# B&R Automation Studio project KeePak_BlissNewScreen (part 2)

#### Cyclic1.st
```iecst
PROGRAM _CYCLIC
	(* Insert code here *)

    // HMI Glue pattern inputs are in inches, but the code needs mm
    gAdhesiveCtrlInterface.Parameters.AdhesivePatterns[0].DelayDistance[0] := gAdhesiveCtrlInterface.Parameters.AdhesiveHMIPatterns[0].DelayDistance[0] * 25.4;
    gAdhesiveCtrlInterface.Parameters.AdhesivePatterns[0].DelayDistance[1] := gAdhesiveCtrlInterface.Parameters.AdhesiveHMIPatterns[0].DelayDistance[1] * 25.4;
    gAdhesiveCtrlInterface.Parameters.AdhesivePatterns[0].DelayDistance[2] := gAdhesiveCtrlInterface.Parameters.AdhesiveHMIPatterns[0].DelayDistance[2] * 25.4;
    gAdhesiveCtrlInterface.Parameters.AdhesivePatterns[0].DelayDistance[3] := gAdhesiveCtrlInterface.Parameters.AdhesiveHMIPatterns[0].DelayDistance[3] * 25.4;
    gAdhesiveCtrlInterface.Parameters.AdhesivePatterns[1].DelayDistance[0] := gAdhesiveCtrlInterface.Parameters.AdhesiveHMIPatterns[1].DelayDistance[0] * 25.4;
    gAdhesiveCtrlInterface.Parameters.AdhesivePatterns[1].DelayDistance[1] := gAdhesiveCtrlInterface.Parameters.AdhesiveHMIPatterns[1].DelayDistance[1] * 25.4;
    gAdhesiveCtrlInterface.Parameters.AdhesivePatterns[1].DelayDistance[2] := gAdhesiveCtrlInterface.Parameters.AdhesiveHMIPatterns[1].DelayDistance[2] * 25.4;
    gAdhesiveCtrlInterface.Parameters.AdhesivePatterns[1].DelayDistance[3] := gAdhesiveCtrlInterface.Parameters.AdhesiveHMIPatterns[1].DelayDistance[3] * 25.4;
    gAdhesiveCtrlInterface.Parameters.AdhesivePatterns[2].DelayDistance[0] := gAdhesiveCtrlInterface.Parameters.AdhesiveHMIPatterns[2].DelayDistance[0] * 25.4;
    gAdhesiveCtrlInterface.Parameters.AdhesivePatterns[2].DelayDistance[1] := gAdhesiveCtrlInterface.Parameters.AdhesiveHMIPatterns[2].DelayDistance[1] * 25.4;
    gAdhesiveCtrlInterface.Parameters.AdhesivePatterns[2].DelayDistance[2] := gAdhesiveCtrlInterface.Parameters.AdhesiveHMIPatterns[2].DelayDistance[2] * 25.4;
    gAdhesiveCtrlInterface.Parameters.AdhesivePatterns[2].DelayDistance[3] := gAdhesiveCtrlInterface.Parameters.AdhesiveHMIPatterns[2].DelayDistance[3] * 25.4;
    gAdhesiveCtrlInterface.Parameters.AdhesivePatterns[3].DelayDistance[0] := gAdhesiveCtrlInterface.Parameters.AdhesiveHMIPatterns[3].DelayDistance[0] * 25.4;
    gAdhesiveCtrlInterface.Parameters.AdhesivePatterns[3].DelayDistance[1] := gAdhesiveCtrlInterface.Parameters.AdhesiveHMIPatterns[3].DelayDistance[1] * 25.4;
    gAdhesiveCtrlInterface.Parameters.AdhesivePatterns[3].DelayDistance[2] := gAdhesiveCtrlInterface.Parameters.AdhesiveHMIPatterns[3].DelayDistance[2] * 25.4;
    gAdhesiveCtrlInterface.Parameters.AdhesivePatterns[3].DelayDistance[3] := gAdhesiveCtrlInterface.Parameters.AdhesiveHMIPatterns[3].DelayDistance[3] * 25.4;

    gAdhesiveCtrlInterface.Parameters.AdhesivePatterns[0].GlueOnDistance[0] := gAdhesiveCtrlInterface.Parameters.AdhesiveHMIPatterns[0].GlueOnDistance[0] * 25.4;
    gAdhesiveCtrlInterface.Parameters.AdhesivePatterns[0].GlueOnDistance[1] := gAdhesiveCtrlInterface.Parameters.AdhesiveHMIPatterns[0].GlueOnDistance[1] * 25.4;
    gAdhesiveCtrlInterface.Parameters.AdhesivePatterns[0].GlueOnDistance[2] := gAdhesiveCtrlInterface.Parameters.AdhesiveHMIPatterns[0].GlueOnDistance[2] * 25.4;
    gAdhesiveCtrlInterface.Parameters.AdhesivePatterns[0].GlueOnDistance[3] := gAdhesiveCtrlInterface.Parameters.AdhesiveHMIPatterns[0].GlueOnDistance[3] * 25.4;
    gAdhesiveCtrlInterface.Parameters.AdhesivePatterns[1].GlueOnDistance[0] := gAdhesiveCtrlInterface.Parameters.AdhesiveHMIPatterns[1].GlueOnDistance[0] * 25.4;
    gAdhesiveCtrlInterface.Parameters.AdhesivePatterns[1].GlueOnDistance[1] := gAdhesiveCtrlInterface.Parameters.AdhesiveHMIPatterns[1].GlueOnDistance[1] * 25.4;
    gAdhesiveCtrlInterface.Parameters.AdhesivePatterns[1].GlueOnDistance[2] := gAdhesiveCtrlInterface.Parameters.AdhesiveHMIPatterns[1].GlueOnDistance[2] * 25.4;
    gAdhesiveCtrlInterface.Parameters.AdhesivePatterns[1].GlueOnDistance[3] := gAdhesiveCtrlInterface.Parameters.AdhesiveHMIPatterns[1].GlueOnDistance[3] * 25.4;
    gAdhesiveCtrlInterface.Parameters.AdhesivePatterns[2].GlueOnDistance[0] := gAdhesiveCtrlInterface.Parameters.AdhesiveHMIPatterns[2].GlueOnDistance[0] * 25.4;
    gAdhesiveCtrlInterface.Parameters.AdhesivePatterns[2].GlueOnDistance[1] := gAdhesiveCtrlInterface.Parameters.AdhesiveHMIPatterns[2].GlueOnDistance[1] * 25.4;
    gAdhesiveCtrlInterface.Parameters.AdhesivePatterns[2].GlueOnDistance[2] := gAdhesiveCtrlInterface.Parameters.AdhesiveHMIPatterns[2].GlueOnDistance[2] * 25.4;
    gAdhesiveCtrlInterface.Parameters.AdhesivePatterns[2].GlueOnDistance[3] := gAdhesiveCtrlInterface.Parameters.AdhesiveHMIPatterns[2].GlueOnDistance[3] * 25.4;
    gAdhesiveCtrlInterface.Parameters.AdhesivePatterns[3].GlueOnDistance[0] := gAdhesiveCtrlInterface.Parameters.AdhesiveHMIPatterns[3].GlueOnDistance[0] * 25.4;
    gAdhesiveCtrlInterface.Parameters.AdhesivePatterns[3].GlueOnDistance[1] := gAdhesiveCtrlInterface.Parameters.AdhesiveHMIPatterns[3].GlueOnDistance[1] * 25.4;
    gAdhesiveCtrlInterface.Parameters.AdhesivePatterns[3].GlueOnDistance[2] := gAdhesiveCtrlInterface.Parameters.AdhesiveHMIPatterns[3].GlueOnDistance[2] * 25.4;
    gAdhesiveCtrlInterface.Parameters.AdhesivePatterns[3].GlueOnDistance[3] := gAdhesiveCtrlInterface.Parameters.AdhesiveHMIPatterns[3].GlueOnDistance[3] * 25.4;

    //SAFETY CHECKS 0001
    IF NOT gAlarmSystemActive THEN
        RETURN;
    END_IF

    //AIR PRESSURE ON/NOK 0002
    //Do not set air pressure alarm unless air pressure has been low for 20 seconds
    AirPressureNotOKTimer.PT := T#20s;
    AirPressureNotOKTimer.IN := (NOT gIO.DIs.AirPressureOK AND NOT gIsSimulated);
    AirPressureNotOKTimer();
    AirPressureNotOK         := AirPressureNotOKTimer.Q;

    //MP ALARMX CHECK STATE AIR PRESSURE LOW 0003
    AirPressureAlarmActive := MpAlarmXCheckState(gAlarmXCore, ALARM_AIR_PRESSURE_LOW, mpALARMX_STATE_ACTIVE);

    //MP ALARMX SET/RESET AIR PRESSURE LOW 0004 AND 0005
    //Set/clear air pressure alarm
    IF (AirPressureNotOK AND NOT AirPressureAlarmActive) THEN
        status := MpAlarmXSet(gAlarmXCore,ALARM_AIR_PRESSURE_LOW);
    ELSIF (NOT AirPressureNotOK AND AirPressureAlarmActive) THEN
        status := MpAlarmXReset(gAlarmXCore,ALARM_AIR_PRESSURE_LOW);
    END_IF

    //MP ALARMX CHECK STATE SAFETY OK/NOK 0006
    SafetyNotOKActive := MpAlarmXCheckState(gAlarmXCore, ALARM_SAFETY_NOTOK, mpALARMX_STATE_ACTIVE);

    //MP ALARMX SET/RESET SAFETY OK/NOK 0007 AND 0008
    //Set/Clear Safety Alarm
    IF (NOT gIO.DIs.SafetyOK AND NOT SafetyNotOKActive AND gIO.SafetyStatus.SafetyProgramRunning) THEN
        status := MpAlarmXSet(gAlarmXCore,ALARM_SAFETY_NOTOK);
    ELSIF (gIO.DIs.SafetyOK AND SafetyNotOKActive AND gIO.SafetyStatus.SafetyProgramRunning) THEN
        status := MpAlarmXReset(gAlarmXCore,ALARM_SAFETY_NOTOK);
    END_IF

    //MP ALARMX CHECK STATE GUARD DOOR 0009
    GuardDoorNotOKActive := MpAlarmXCheckState(gAlarmXCore, ALARM_SAFETY_GUARD_DOOR, mpALARMX_STATE_ACTIVE);

    //MP ALARMX SET/RESET GUARD DOORS 0010 AND 0011
    //Set/Clear Safety Alarm
    IF (NOT gIO.SafetyStatus.GuardDoorsOK AND NOT GuardDoorNotOKActive AND gIO.SafetyStatus.SafetyProgramRunning) THEN
        status := MpAlarmXSet(gAlarmXCore,ALARM_SAFETY_GUARD_DOOR);
    ELSIF (gIO.SafetyStatus.GuardDoorsOK AND GuardDoorNotOKActive AND gIO.SafetyStatus.SafetyProgramRunning) THEN
        status := MpAlarmXReset(gAlarmXCore,ALARM_SAFETY_GUARD_DOOR);
    END_IF

    //MP ALARMX CHECK STATE FRONT ESTOP 0012
    FrontEStopNotOKActive := MpAlarmXCheckState(gAlarmXCore, ALARM_SAFETY_FRONT_ESTOP, mpALARMX_STATE_ACTIVE);

    //MP ALARMX SET/RESET FRONT ESTOP 0013 AND 0014
    //Set/Clear Safety Alarm
    IF (NOT gIO.SafetyStatus.FrontEStopOK AND NOT FrontEStopNotOKActive AND gIO.SafetyStatus.SafetyProgramRunning) THEN
        status := MpAlarmXSet(gAlarmXCore,ALARM_SAFETY_FRONT_ESTOP);
    ELSIF (gIO.SafetyStatus.FrontEStopOK AND FrontEStopNotOKActive AND gIO.SafetyStatus.SafetyProgramRunning) THEN
        status := MpAlarmXReset(gAlarmXCore,ALARM_SAFETY_FRONT_ESTOP);
    END_IF

    //MP ALARMX CHECK STATE REAR ESTOP 0015
    RearEStopNotOKActive := MpAlarmXCheckState(gAlarmXCore, ALARM_SAFETY_REAR_ESTOP, mpALARMX_STATE_ACTIVE);

    //MP ALARMX SET/RESET REAR ESTOP 0016 AND 0017
    //Set/Clear Safety Alarm
    IF (NOT gIO.SafetyStatus.BackEstopOK AND NOT RearEStopNotOKActive AND gIO.SafetyStatus.SafetyProgramRunning) THEN
        status := MpAlarmXSet(gAlarmXCore,ALARM_SAFETY_REAR_ESTOP);
    ELSIF (gIO.SafetyStatus.BackEstopOK AND RearEStopNotOKActive AND gIO.SafetyStatus.SafetyProgramRunning) THEN
        status := MpAlarmXReset(gAlarmXCore,ALARM_SAFETY_REAR_ESTOP);
    END_IF

    //TURN AIR ON 0018
    //If safety is OK, Turn air On and turn off the red light
    gIO.DOs.AirOn         := gIO.DIs.SafetyOK;
    gIO.DOs.RedLightStack := NOT (gIO.DIs.SafetyOK AND NOT gModeControlInterface.Status.BlissPanelAlarmActive);

    //NO ALARMS GREEN LIGHT 0019
    //If there are no alarms active, turn on the green light
    gIO.DOs.GreenLightStack := NOT gAlarmActive;

    //ALARM YELLOW LIGHT 0020
    //If there is an active alarm, or the hopper is low, turn on yellow stack light
    gIO.DOs.AmberLightStack := (gAlarmActive OR gIO.DIs.BodyHopperLow);

	//DO NOT FINISH CYCLE OF ANYTHING OTHER THAN STOP BUTTON IS PRESSED 0024
	//If an alarm is active or safety is not ok or jog mode is selected, do not finish the selected cycle
	IF (gServoFeedInterface.Status.Error OR gBodyHopperInterface.Status.Error OR gLeftHopperInterface.Status.Error OR gRightHopperInterface.Status.Error OR gServoRamInterface.Status.Error OR
		NOT gIO.DIs.SafetyOK OR gHMI.Commands.SelectJogMode OR gHighSeverityAlarmActive OR BodyCheckError) THEN
		PickAndPlaceHasBox                         := FALSE;
		PickAndPlaceDwelling                       := FALSE;
		PhotoEyeSeen                               := FALSE;
		Vacuum_ON                                  := FALSE;
		gIO.DOs.X_PickSolenoid                     := FALSE;
		gIO.DOs.BlowOffOn                          := FALSE;
	END_IF

	//DOES NOT LET MACHINE RUN IF GLUE SYSTEM HAS AN ERROR 0025
	//Do not allow machine to run if glue system has an alarm (Removed gLowSeverityAlarmActive)
	IF (gAdhesiveCtrlInterface.Status.AlarmActive OR
		gServoFeedInterface.Status.Error OR gBodyHopperInterface.Status.Error OR gLeftHopperInterface.Status.Error OR gRightHopperInterface.Status.Error OR gServoRamInterface.Status.Error OR
		gLowSeverityAlarmActive OR gHighSeverityAlarmActive OR gServoPnPInterface.Status.Error) THEN
		gHMI.Commands.RequestVFDRun := FALSE;
	END_IF

	//AUTO MODE RUN REQUEST FINISH CYCLE 0026
	//If we're in auto mode, and run request has been made or we should finish the running, set move request
	MoveVelocityRequest := (gHMI.Commands.SelectAutoMode AND gHMI.Commands.RequestVFDRun);

	//RAM POSITION AND STOP POSITION (360-0 ROLLOVER)DetermineDistanceToStopPos 0027
	DistanceFromStopPosition := DetermineDistanceToStopPos(gIO.Encoders.FeedEncoderPos, gModeControlInterface.Parameters.StopPosition);

	//KEEPS SERVOS RUNNING TO FINISH CYCLE 0030
	//VFD run command was the run command for the old machine. Keep servos cycling while it is true
	gHMI.Commands.StartBodyHopper := gHMI.Commands.RequestVFDRun;
	gHMI.Commands.StartLeftHopper := gHMI.Commands.RequestVFDRun;
	gHMI.Commands.StartRightHopper := gHMI.Commands.RequestVFDRun;
	gHMI.Commands.StartServoFeed   := (gHMI.Commands.RequestVFDRun (*AND NOT DownstreamBlocked*) AND NOT StopFeedServo);
	gHMI.Commands.CycleServoRam    := gHMI.Commands.RequestVFDRun;
	gHMI.Commands.CycleServoPnP    := gHMI.Commands.RequestVFDRun;
	// The discharge conveyor is controlled by three bits.
	// If #1 is on, then it is running slow. If #1 and #3 are on, then it is running medium speed. #2 Can be used if we need a faster speed.
	gIO.DOs.OutConveyorOn_1 := gHMI.Commands.RequestVFDRun OR (gCyclesToFinish > 0);
	gIO.DOs.OutConveyorOn_2 := gHMI.Commands.RequestVFDRun OR (gCyclesToFinish > 0);
	gIO.DOs.OutConveyorOn_3 := gHMI.Commands.RequestVFDRun OR (gCyclesToFinish > 0);

	//RISING EDGE FOR SERVOINPUT SIGNAL 0031
	Rtrig_FeedServoTMR(CLK := FeedServoTMR.Q);
	StopFeed := Rtrig_FeedServoTMR.Q;

	//0032 SERVO RAM TRIGGER SET IN FEED HANDLER. COMMENTED OUT

	//HOPPER LOW ALARMS 0033
	BodyHopperLowTMR.IN := gIO.DIs.BodyHopperLow;
    BodyHopperLowTMR.PT := gHMI.Parameters.LowBodyHopperTime;
    BodyHopperLowTMR();
    IF BodyHopperLowTMR.Q THEN
        BodyHopperLowAlarm := TRUE;
	END_IF
	LeftHopperLowTMR.IN := gIO.DIs.LeftHopperLow;
	LeftHopperLowTMR.PT := gHMI.Parameters.LowLeftHopperTime;
	LeftHopperLowTMR();
	IF LeftHopperLowTMR.Q THEN
		LeftHopperLowAlarm := TRUE;
	END_IF
	RightHopperLowTMR.IN := gIO.DIs.RightHopperLow;
	RightHopperLowTMR.PT := gHMI.Parameters.LowRightHopperTime;
	RightHopperLowTMR();
	IF RightHopperLowTMR.Q THEN
		RightHopperLowAlarm := TRUE;
	END_IF

    //FEED STOP TIMER 0034
    //Timer for the HopperLows to trigger StopFeed
    FeedStopTimer.IN := gIO.DIs.BodyHopperLow OR gIO.DIs.RightHopperLow OR gIO.DIs.LeftHopperLow;
    FeedStopTimer.PT := gHMI.Parameters.LowHopperTime;
    FeedStopTimer();
    HoperLowStop     := FeedStopTimer.Q;

    //HOPPER LOW ALARM RESET 0035
    IF NOT gIO.DIs.BodyHopperLow THEN
        BodyHopperLowAlarm := FALSE;
	END_IF
	IF NOT gIO.DIs.LeftHopperLow THEN
		LeftHopperLowAlarm := FALSE;
	END_IF
	IF NOT gIO.DIs.RightHopperLow THEN
		RightHopperLowAlarm := FALSE;
	END_IF

	//==========================================================================================================================================================
	//==========================================================================================================================================================

	//PHOTO EYES SETTING AND RESETTING
	IF (gIO.DIs.AdhesivePhotoEye) THEN
		PhotoEyeSeen := TRUE;
	END_IF
    IF gIO.DIs.BodyDetect THEN
        PhotoEyeSeen := FALSE;
    END_IF

    //0047
    //Latch the encoder position. this marks the start of the glue cycle
    Rtrig_PhotoEyeSeen(CLK := PhotoEyeSeen);
    IF (Rtrig_PhotoEyeSeen.Q AND ((gHMI.Commands.SelectAutoMode AND gHMI.Commands.RequestVFDRun) OR (gCyclesToFinish > 0))) THEN
        gAdhesiveCtrlInterface.Status.LatchedEncoderPos := LREAL_TO_REAL(gServoFeedInterface.Status.ActualPosition);
        DistanceAfterLatch                              := 0;
        OldEncoderPos                                   := LREAL_TO_REAL(gServoFeedInterface.Status.ActualPosition);
    END_IF

    //0048
    //Determine how far the ram has moved since the photo eye was last seen
    DistanceAfterLatch := (ComputeDistanceMoved(LREAL_TO_REAL(gServoFeedInterface.Status.ActualPosition),OldEncoderPos) + DistanceAfterLatch);

    //0049
    OldEncoderPos := LREAL_TO_REAL(gServoFeedInterface.Status.ActualPosition);

	//BODY PANEL TIMEOUT 0052
	//If the machine is running and a box has passed the photoeyes, but hasn't cleared the photo eye for LowFeedJamTime amount of time, then raise an alarm
    BodyPanelTimeout.PT := gHMI.Parameters.LowFeedJamTime;
    BodyPanelTimeout.IN := (gHMI.Commands.RequestVFDRun AND gIO.DIs.BodyDetect);
    BodyPanelTimeout();
    IF BodyPanelTimeout.Q THEN
        BodyCheckError := TRUE;
    ELSIF gHMI.Commands.RequestReset THEN
        BodyCheckError := FALSE;
	END_IF

	//INFEED TIMEOUT
	//If the machine is running and a box hasnt passed the photoeyes for LowFeedJamTime amount of time, then raise an alarm
	InfeedTimeout.PT := gHMI.Parameters.TopFeedJamTime;
	InfeedTimeout.IN := (gHMI.Commands.RequestVFDRun AND NOT gIO.DIs.BodyDetect);
	InfeedTimeout();
	IF InfeedTimeout.Q THEN
		InfeedCheckError := TRUE;
	ELSIF gHMI.Commands.RequestReset THEN
		InfeedCheckError := FALSE;
	END_IF

    //0053 AND 0054 LUBE COUNTER
    LubricationOK := (LubeCount < gHMI.Parameters.SetCycleCount);

    Rtrig_LubricationCounter(CLK := gIO.DIs.LubricationCounter);
    LubricationCounter.CU    := Rtrig_LubricationCounter.Q;
    LubricationCounter.RESET := LubeReset;
    LubricationCounter.PV    := UDINT_TO_UINT(gHMI.Parameters.LubeCycleCount);
    LubricationCounter();
    CountReset               := LubricationCounter.Q;

    //0055 COUNT AND LUBE COUNT RESET
    LubeReset := CountReset;
    IF CountReset THEN
        LubeCount := 0;
	END_IF

	//make it a fault if the system is reuqested to run while any hopper is off
	IF gHMI.Commands.RequestVFDRun AND (gIO.DIs.LeftHopperMotor_OFF OR gIO.DIs.RightHopperMotor_OFF OR gIO.DIs.BodyHopperMotor_OFF) THEN
		HopperRunningError := TRUE;
	ELSIF gHMI.Commands.RequestReset THEN
		HopperRunningError := FALSE;
	END_IF

    //Disabled this due to the error triggering and not clearing after a few hours
//    PnPTimeout.PT := T#3600s;
//    PnPTimeout.IN := NOT gHMI.Commands.RequestVFDRun AND (gHMI.Commands.RequestStop OR gServoPnPInterface.Status.PoweredOn);
//    PnPTimeout();
 //   IF PnPTimeout.Q THEN
//        PnPTimeoutError := TRUE;
//    ELSIF gHMI.Commands.RequestReset THEN
//        PnPTimeoutError := FALSE;
//    END_IF

	END_PROGRAM
```

### Variables.var
```iecst
VAR
	StartDwellTimer : TON;
	AtTorqueTimer : TON;
	state : ServoHopperState_enum;
END_VAR
VAR RETAIN
	CycleCount : UDINT;
END_VAR
VAR
	ResetTimeoutAlarm : BOOL;
	ResetTimeoutTimer : TON;
END_VAR
```

### Program Logical/ServoMotion/LeftHopperHandler

#### Main.st
```iecst
PROGRAM _INIT
	(* Insert code here *)

	gHMI.Parameters.LeftHopperJogVelocity := 3.35;
	gHMI.Parameters.LeftHopperVelocity := 3.35;
	gHMI.Parameters.LeftHopperAccel := 180.0;

	gHMI.Parameters.LeftHopperTorqueLimit := 1.0;

	gHMI.Parameters.LeftHopperDwellTime := 1500; //1 s
	gHMI.Parameters.AtTorqueTime := 500; //1 s

	gHMI.Parameters.LeftHopperTimeoutTime := 600000; //10 minutes

END_PROGRAM

PROGRAM _CYCLIC

	IF gNumActiveAlarms  > 0 THEN
		state := SERVOHOPPER_ERROR;
	END_IF

	IF gHighSeverityAlarmActive THEN
		state := SERVOHOPPER_ERROR;
	END_IF

	//make sure that torque limiting is turned on while jogging
	//	IF EDGEPOS(gHMI.Commands.JogLeftHopperPos) THEN
	//		gLeftHopperInterface.Commands.ToMapp.TorqueLimitingOn := TRUE;
	//	END_IF
	//	IF EDGEPOS(gHMI.Commands.JogLeftHopperNeg) THEN
	//		gLeftHopperInterface.Commands.ToMapp.TorqueLimitingOn := TRUE;
	//	END_IF

	StartDwellTimer.IN := FALSE; //clear otuside state machine. will be set true in appropriate state
	AtTorqueTimer.IN := FALSE;
	ResetTimeoutTimer.IN := FALSE;

	// If the hopper has been reset but the machine isn't running, only let the hopper run for an alotted time to protect the motor
	IF gIO.DIs.LeftHopperMotor_RUN AND NOT gLeftHopperInterface.Status.Error AND (NOT gHMI.Commands.RequestVFDRun) THEN
		ResetTimeoutTimer.IN := TRUE;
	END_IF
	IF ResetTimeoutTimer.Q THEN
		ResetTimeoutAlarm := TRUE;
	END_IF

	// Resetting clears the timeout alarms
	IF gHMI.Commands.RequestReset THEN
		ResetTimeoutAlarm := FALSE;
	END_IF

	CASE state OF

		SERVOHOPPER_WAIT_FOR_HOME:

			//servo ram should home automatically on machine start up. This is a direct home axis and should not rquire a home command
			IF gServoFeedInterface.Status.Homed THEN
				gLeftHopperInterface.Commands.ToMapp.TorqueLimitingOn := TRUE;
				state := SERVOHOPPER_IDLE;
			END_IF

		SERVOHOPPER_IDLE:

			IF gIO.DIs.LeftHopperMotor_RUN AND LeftHopperFirstHomeExecuted THEN
				gLeftHopperInterface.Commands.ToMapp.TorqueLimitingOn := TRUE; //turn torque limiting on

				gLeftHopperInterface.Commands.RequestMoveVelocity := TRUE;
				gLeftHopperInterface.Parameters.MovementParameters.Direction := 0;

				state := SERVOHOPPER_MOVE_VELOCITY;
			END_IF

		SERVOHOPPER_MOVE_VELOCITY:

			AtTorqueTimer.IN := (gLeftHopperInterface.Status.ActualTorque >= gHMI.Parameters.LeftHopperTorqueLimit *0.90);

			IF gIO.DIs.LeftHopperMotor_OFF = TRUE THEN
				gLeftHopperInterface.Commands.RequestMoveVelocity := FALSE;
				state := SERVOHOPPER_IDLE;
			ELSIF AtTorqueTimer.Q THEN
				gLeftHopperInterface.Parameters.MovementParameters.Direction := 1;
				gLeftHopperInterface.Commands.ToMapp.Update := TRUE;
				gLeftHopperInterface.Commands.RequestMoveVelocity := TRUE;
				state := SERVOHOPPER_COOLDOWN;
			END_IF

		SERVOHOPPER_COOLDOWN:

			StartDwellTimer.IN := TRUE;

			IF gIO.DIs.LeftHopperMotor_OFF = TRUE THEN
				gLeftHopperInterface.Commands.RequestMoveVelocity := FALSE;
				state := SERVOHOPPER_IDLE;
			ELSIF StartDwellTimer.Q THEN
				gLeftHopperInterface.Parameters.MovementParameters.Direction := 0;
				gLeftHopperInterface.Commands.ToMapp.Update := TRUE;
				gLeftHopperInterface.Commands.RequestMoveVelocity := TRUE;
				state := SERVOHOPPER_MOVE_VELOCITY;
			END_IF

		SERVOHOPPER_ERROR:

			gLeftHopperInterface.Status.MoveComplete := TRUE;
			gHMI.Commands.StartLeftHopper := FALSE;

			gLeftHopperInterface.Commands.RequestMoveVelocity := FALSE;

			ResetTimeoutTimer.IN := FALSE;

			IF (gNumActiveAlarms = 0) THEN
				state := SERVOHOPPER_WAIT_FOR_HOME;
			END_IF

	END_CASE;

	StartDwellTimer.PT := gHMI.Parameters.LeftHopperDwellTime; //500 ms
	StartDwellTimer();
	AtTorqueTimer.PT := gHMI.Parameters.AtTorqueTime; //500 ms
	AtTorqueTimer();
	ResetTimeoutTimer.PT := gHMI.Parameters.LeftHopperTimeoutTime;
	ResetTimeoutTimer();

END_PROGRAM

PROGRAM _EXIT
				(* Insert code here *)

END_PROGRAM
```

### Program Logical/ServoMotion/MappCalls

#### Cyclic.ld
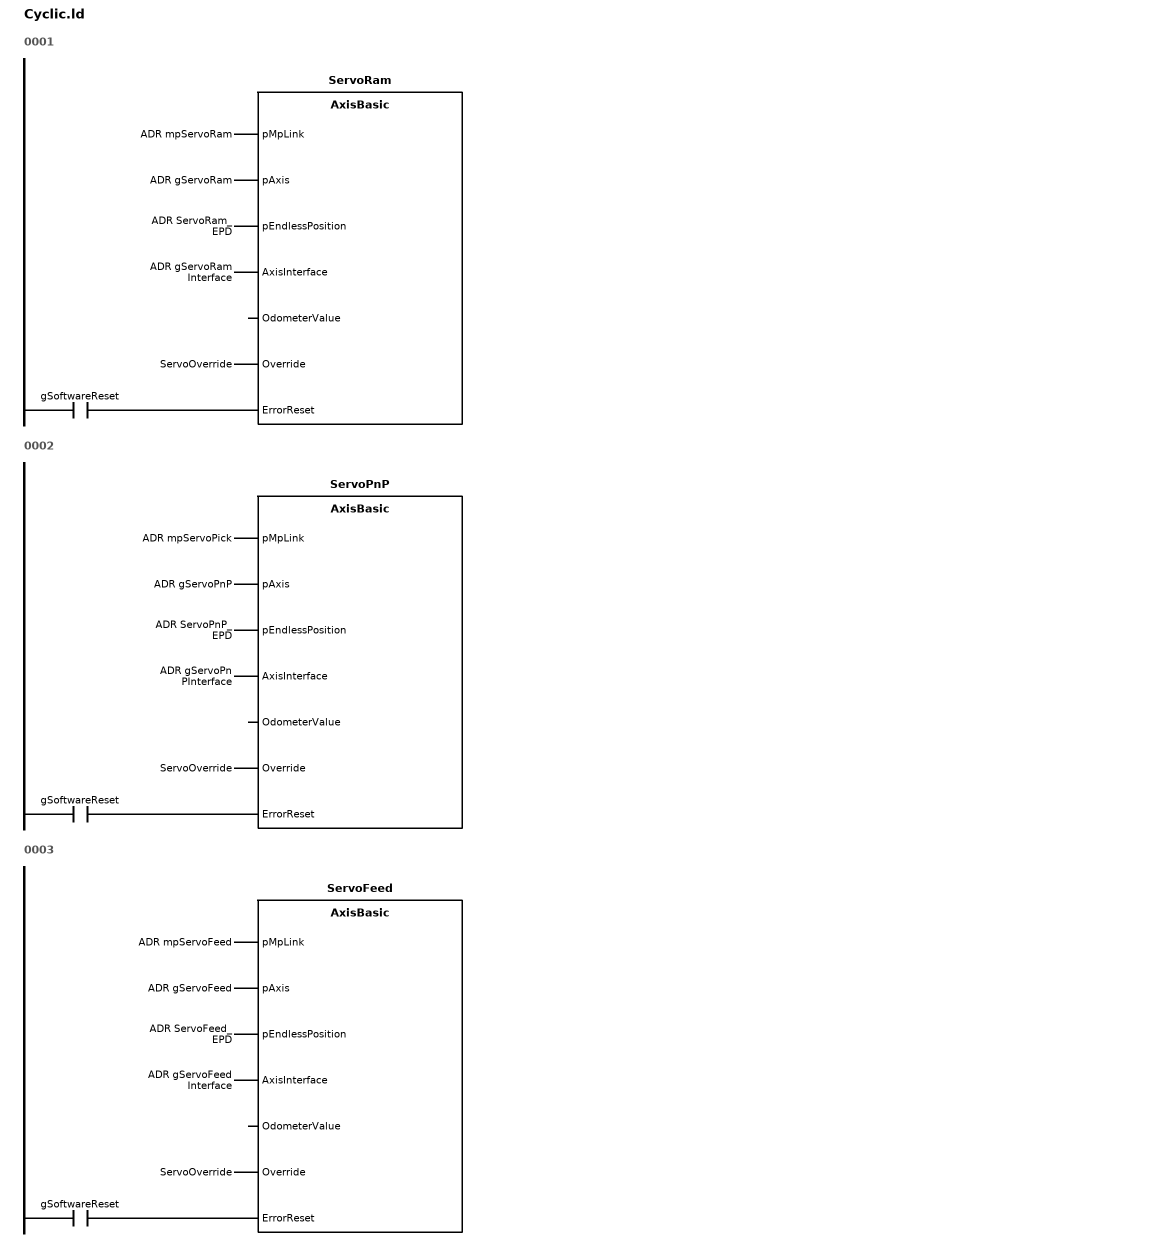
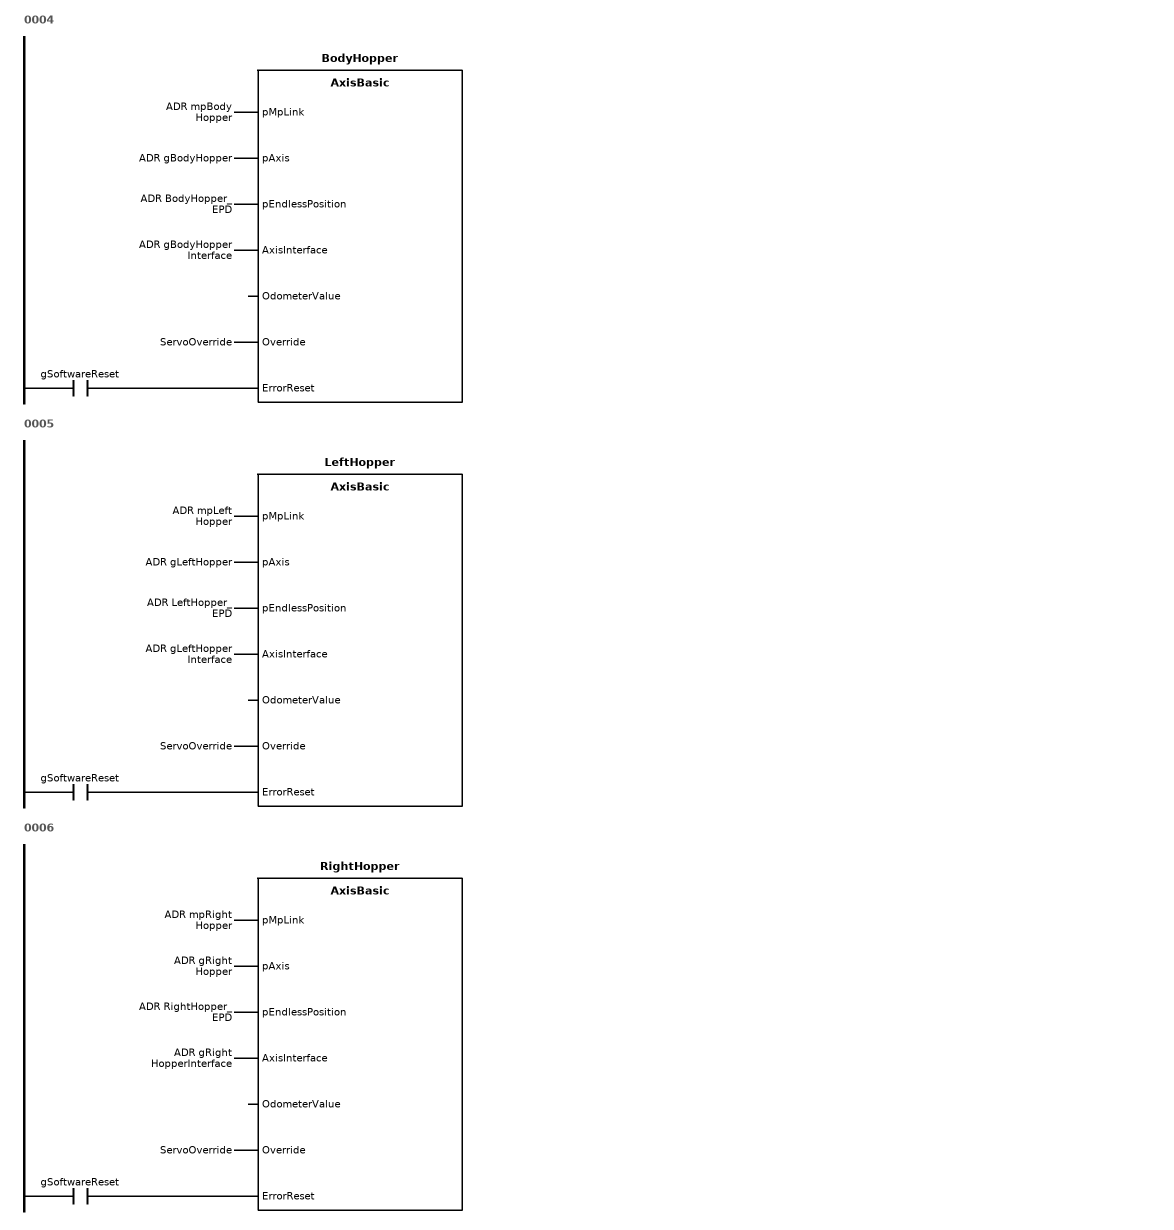
Ladder, written as Structured Text:
```iecst
PROGRAM _CYCLIC
(* Network 1 *)
ServoRam(pMpLink := ADR(mpServoRam), pAxis := ADR(gServoRam), pEndlessPosition := ADR(ServoRam_EPD), AxisInterface := ADR(gServoRamInterface), Override := ServoOverride, ErrorReset := gSoftwareReset);

(* Network 2 *)
ServoPnP(pMpLink := ADR(mpServoPick), pAxis := ADR(gServoPnP), pEndlessPosition := ADR(ServoPnP_EPD), AxisInterface := ADR(gServoPnPInterface), Override := ServoOverride, ErrorReset := gSoftwareReset);

(* Network 3 *)
ServoFeed(pMpLink := ADR(mpServoFeed), pAxis := ADR(gServoFeed), pEndlessPosition := ADR(ServoFeed_EPD), AxisInterface := ADR(gServoFeedInterface), Override := ServoOverride, ErrorReset := gSoftwareReset);

(* Network 4 *)
BodyHopper(pMpLink := ADR(mpBodyHopper), pAxis := ADR(gBodyHopper), pEndlessPosition := ADR(BodyHopper_EPD), AxisInterface := ADR(gBodyHopperInterface), Override := ServoOverride, ErrorReset := gSoftwareReset);

(* Network 5 *)
LeftHopper(pMpLink := ADR(mpLeftHopper), pAxis := ADR(gLeftHopper), pEndlessPosition := ADR(LeftHopper_EPD), AxisInterface := ADR(gLeftHopperInterface), Override := ServoOverride, ErrorReset := gSoftwareReset);

(* Network 6 *)
RightHopper(pMpLink := ADR(mpRightHopper), pAxis := ADR(gRightHopper), pEndlessPosition := ADR(RightHopper_EPD), AxisInterface := ADR(gRightHopperInterface), Override := ServoOverride, ErrorReset := gSoftwareReset);
END_PROGRAM
```

### Program Logical/ServoMotion/MotionHandler

#### Variables.var
```iecst
VAR
	ServoFeedHandler : AxisHandler;
	ServoPnPHandler : AxisHandler;
	BodyHopperHandler : AxisHandler;
	LeftHopperHandler : AxisHandler;
	RightHopperHandler : AxisHandler;
	ServoRamHandler : AxisHandler;
	OldTorqueLimitBodyHopper : REAL;
	OldTorqueLimitLeftHopper : REAL;
	OldTorqueLimitRightHopper : REAL;
	OldTorqueLimitFeed : REAL;
	OldTorqueLimitRam : REAL;
	SetHardwareInputs : MC_BR_SetHardwareInputs;
END_VAR
```

#### Main.c
```c
#include <bur/plctypes.h>

#ifdef _DEFAULT_INCLUDES
#include <AsDefault.h>
#endif

/**
* This task:
*
* Populates homing and coupling defaults for each axis
* Instantiates axis control state machines for each axis
*
*
*/

void _INIT ProgramInit(void)
{

	gHomingParameters.ServoRam.Mode = mpAXIS_HOME_MODE_BLOCK_DS; //Servo Ram homes to hard stop
	gHomingParameters.ServoRam.BlockDetectionPositionError = 1.5;
	gHomingParameters.ServoRam.PositionErrorStopLimit = 2.0;
	gHomingParameters.ServoRam.StartDirection = mpAXIS_HOME_DIR_NEGATIVE;
	gHomingParameters.ServoRam.HomingDirection = mpAXIS_HOME_DIR_POSITIVE;
	gHomingParameters.ServoRam.StartVelocity = 10;
	gHomingParameters.ServoRam.HomingVelocity = 5;
	gHomingParameters.ServoRam.Position = 0.5;
	gHomingParameters.ServoRam.SensorOffset = 12.5; //back off switch by 12.5 mm and call that position home
	gHomingParameters.ServoRam.TorqueLimit = 2.0;

	gHomingParameters.ServoPnP.Mode = mpAXIS_HOME_MODE_ABS_SWITCH; // Pick and place homes to a switch
	gHomingParameters.ServoPnP.SwitchEdge = mpAXIS_HOME_DIR_NEGATIVE;
	gHomingParameters.ServoPnP.StartDirection = mpAXIS_HOME_DIR_NEGATIVE;
	gHomingParameters.ServoPnP.HomingDirection = mpAXIS_HOME_DIR_POSITIVE;
	gHomingParameters.ServoPnP.StartVelocity = 5;
	gHomingParameters.ServoPnP.HomingVelocity = 5;
	gHomingParameters.ServoPnP.Position = 0;
	gHomingParameters.ServoPnP.SensorOffset = 0;
	gHomingParameters.ServoPnP.TorqueLimit = 3.0;

	gHomingParameters.ServoFeed.Mode = mpAXIS_HOME_MODE_DIRECT;
	gHomingParameters.ServoFeed.StartDirection = mpAXIS_HOME_DIR_NEGATIVE;
	gHomingParameters.ServoFeed.HomingDirection = mpAXIS_HOME_DIR_POSITIVE;
	gHomingParameters.ServoFeed.Position = 0;
	gHomingParameters.ServoFeed.SensorOffset = 0;

	gHomingParameters.BodyHopper.Mode = mpAXIS_HOME_MODE_DIRECT;
	gHomingParameters.BodyHopper.StartDirection = mpAXIS_HOME_DIR_NEGATIVE;
	gHomingParameters.BodyHopper.HomingDirection = mpAXIS_HOME_DIR_POSITIVE;
	gHomingParameters.BodyHopper.Position = 0;
	gHomingParameters.BodyHopper.SensorOffset = 0;

	gHomingParameters.LeftHopper.Mode = mpAXIS_HOME_MODE_DIRECT;
	gHomingParameters.LeftHopper.StartDirection = mpAXIS_HOME_DIR_NEGATIVE;
	gHomingParameters.LeftHopper.HomingDirection = mpAXIS_HOME_DIR_POSITIVE;
	gHomingParameters.LeftHopper.Position = 0;
	gHomingParameters.LeftHopper.SensorOffset = 0;

	gHomingParameters.RightHopper.Mode = mpAXIS_HOME_MODE_DIRECT;
	gHomingParameters.RightHopper.StartDirection = mpAXIS_HOME_DIR_NEGATIVE;
	gHomingParameters.RightHopper.HomingDirection = mpAXIS_HOME_DIR_POSITIVE;
	gHomingParameters.RightHopper.Position = 0;
	gHomingParameters.RightHopper.SensorOffset = 0;

	ServoRamFirstHomeExecuted = 0; //THIS MUST ALWAYS BE SET TO FALSE. THIS IS A SINGLE TURN ENCODER
	ServoPnPFirstHomeExecuted = 0;
	ServoFeedFirstHomeExecuted = 0; //THIS MUST ALWAYS BE SET TO FALSE. THIS IS A SINGLE TURN ENCODER
	BodyHopperFirstHomeExecuted = 0; //THIS MUST ALWAYS BE SET TO FALSE. THIS IS A SINGLE TURN ENCODER
	LeftHopperFirstHomeExecuted = 0; //THIS MUST ALWAYS BE SET TO FALSE. THIS IS A SINGLE TURN ENCODER
	RightHopperFirstHomeExecuted = 0; //THIS MUST ALWAYS BE SET TO FALSE. THIS IS A SINGLE TURN ENCODER

	//******* Start Axis and Drive Param Default Settings *******//

	//ram

	strcpy((char*)&gServoRamInterface.Parameters.AxisAndDrivePars.AxisName, "Ram");
	gServoRamInterface.Parameters.AxisAndDrivePars.Axis.BaseType = mpAXIS_LIMITED_LINEAR;
	gServoRamInterface.Parameters.AxisAndDrivePars.Axis.MeasurementUnit = mpAXIS_UNIT_MM;
	gServoRamInterface.Parameters.AxisAndDrivePars.Axis.MeasurementResolution = 0.01;
	gServoRamInterface.Parameters.AxisAndDrivePars.Axis.SoftwareLimitPositions.LowerLimit = 0;
	gServoRamInterface.Parameters.AxisAndDrivePars.Axis.SoftwareLimitPositions.UpperLimit = 870.0;
	gServoRamInterface.Parameters.AxisAndDrivePars.Axis.PeriodSettings.Period = 360;

	gServoRamInterface.Parameters.AxisAndDrivePars.Axis.MovementLimits.VelocityPositive = 1391.0;
	gServoRamInterface.Parameters.AxisAndDrivePars.Axis.MovementLimits.VelocityNegative = 1391.0;
	gServoRamInterface.Parameters.AxisAndDrivePars.Axis.MovementLimits.Acceleration = 3055.0;
	gServoRamInterface.Parameters.AxisAndDrivePars.Axis.MovementLimits.Deceleration = 3055.0;
	gServoRamInterface.Parameters.AxisAndDrivePars.Axis.MovementLimits.JerkTime = 0.0;
	gServoRamInterface.Parameters.AxisAndDrivePars.Axis.MovementLimits.PositionErrorStopLimit = 12;
	gServoRamInterface.Parameters.AxisAndDrivePars.Axis.MovementLimits.VelocityErrorStopLimit = 0.0;
	gServoRamInterface.Parameters.AxisAndDrivePars.Axis.MovementLimits.VelocityErrorStopLimitMode = mpAXIS_VEL_MODE_OFF;

	//gServoRamInterface.Parameters.AxisAndDrivePars.Axis.CyclicReadChannels.UserChannelParameterID = 214;

	gServoRamInterface.Parameters.AxisAndDrivePars.Drive.Gearbox.Input = 882; //actual gear ratio is 8.82 motor turns per load rev
	gServoRamInterface.Parameters.AxisAndDrivePars.Drive.Gearbox.Output = 100;
	gServoRamInterface.Parameters.AxisAndDrivePars.Drive.Gearbox.Direction = mpAXIS_DIR_COUNTERCLOCKWISE;

	gServoRamInterface.Parameters.AxisAndDrivePars.Drive.Transformation.ReferenceDistance = 245.53333;

	//gServoRamInterface.Parameters.AxisAndDrivePars.Drive.Controller.Mode = mpAXIS_CTRL_MODE_POSITION_FF;
	gServoRamInterface.Parameters.AxisAndDrivePars.Drive.Controller.Mode = mpAXIS_CTRL_MODE_POSITION;
	gServoRamInterface.Parameters.AxisAndDrivePars.Drive.Controller.Position.ProportionalGain = 250.0;
	gServoRamInterface.Parameters.AxisAndDrivePars.Drive.Controller.Position.IntegralTime = 0.0;
	gServoRamInterface.Parameters.AxisAndDrivePars.Drive.Controller.Position.PredictionTime = 0.0004;
	gServoRamInterface.Parameters.AxisAndDrivePars.Drive.Controller.Position.TotalDelayTime = 0.0004;

	gServoRamInterface.Parameters.AxisAndDrivePars.Drive.Controller.Speed.ProportionalGain = 7.5;
	gServoRamInterface.Parameters.AxisAndDrivePars.Drive.Controller.Speed.IntegralTime = 0.1;
	gServoRamInterface.Parameters.AxisAndDrivePars.Drive.Controller.Speed.FilterTime = 0.0;

	//these values are only used if controller mode is set to position + feed forward
	gServoRamInterface.Parameters.AxisAndDrivePars.Drive.Controller.FeedForward.TorqueLoad = 0.0;
	gServoRamInterface.Parameters.AxisAndDrivePars.Drive.Controller.FeedForward.TorquePositive = 0.0;
	gServoRamInterface.Parameters.AxisAndDrivePars.Drive.Controller.FeedForward.TorqueNegative = 0.0;
	gServoRamInterface.Parameters.AxisAndDrivePars.Drive.Controller.FeedForward.SpeedTorqueFactor = 0.0;
	gServoRamInterface.Parameters.AxisAndDrivePars.Drive.Controller.FeedForward.Inertia = 0.0;
	gServoRamInterface.Parameters.AxisAndDrivePars.Drive.Controller.FeedForward.AccelerationFilterTime = 0.0;

	//pick and place

	strcpy((char*)&gServoPnPInterface.Parameters.AxisAndDrivePars.AxisName, "PickNPlace");
	gServoPnPInterface.Parameters.AxisAndDrivePars.Axis.BaseType = mpAXIS_LIMITED_ROTARY;
	gServoPnPInterface.Parameters.AxisAndDrivePars.Axis.MeasurementUnit = mpAXIS_UNIT_DEGREES;
	gServoPnPInterface.Parameters.AxisAndDrivePars.Axis.MeasurementResolution = 0.01;
	gServoPnPInterface.Parameters.AxisAndDrivePars.Axis.SoftwareLimitPositions.LowerLimit = 0;
	gServoPnPInterface.Parameters.AxisAndDrivePars.Axis.SoftwareLimitPositions.UpperLimit = 115;
	gServoPnPInterface.Parameters.AxisAndDrivePars.Axis.PeriodSettings.Period = 360;

	gServoPnPInterface.Parameters.AxisAndDrivePars.Axis.MovementLimits.VelocityPositive = 1800.0;
	gServoPnPInterface.Parameters.AxisAndDrivePars.Axis.MovementLimits.VelocityNegative = 1800.0;
	gServoPnPInterface.Parameters.AxisAndDrivePars.Axis.MovementLimits.Acceleration = 30800.0;
	gServoPnPInterface.Parameters.AxisAndDrivePars.Axis.MovementLimits.Deceleration = 30800.0;
	gServoPnPInterface.Parameters.AxisAndDrivePars.Axis.MovementLimits.JerkTime = 0.0;
	gServoPnPInterface.Parameters.AxisAndDrivePars.Axis.MovementLimits.PositionErrorStopLimit = 4;
	gServoPnPInterface.Parameters.AxisAndDrivePars.Axis.MovementLimits.VelocityErrorStopLimit = 2;
	gServoPnPInterface.Parameters.AxisAndDrivePars.Axis.MovementLimits.VelocityErrorStopLimitMode = mpAXIS_VEL_MODE_OFF;

	//gServoPnPInterface.Parameters.AxisAndDrivePars.Axis.CyclicReadChannels.UserChannelParameterID = 214;

	gServoPnPInterface.Parameters.AxisAndDrivePars.Drive.Gearbox.Input = 10;
	gServoPnPInterface.Parameters.AxisAndDrivePars.Drive.Gearbox.Output = 1;
	gServoPnPInterface.Parameters.AxisAndDrivePars.Drive.Gearbox.Direction = mpAXIS_DIR_CLOCKWISE;

	gServoPnPInterface.Parameters.AxisAndDrivePars.Drive.Transformation.ReferenceDistance = 360;

	//gServoPnPInterface.Parameters.AxisAndDrivePars.Drive.Controller.Mode = mpAXIS_CTRL_MODE_POSITION_FF;
	gServoPnPInterface.Parameters.AxisAndDrivePars.Drive.Controller.Mode = mpAXIS_CTRL_MODE_POSITION;
	gServoPnPInterface.Parameters.AxisAndDrivePars.Drive.Controller.Position.ProportionalGain = 600.0;
	gServoPnPInterface.Parameters.AxisAndDrivePars.Drive.Controller.Position.IntegralTime = 0.0;
	gServoPnPInterface.Parameters.AxisAndDrivePars.Drive.Controller.Position.PredictionTime = 0.0004;
	gServoPnPInterface.Parameters.AxisAndDrivePars.Drive.Controller.Position.TotalDelayTime = 0.0004;

	gServoPnPInterface.Parameters.AxisAndDrivePars.Drive.Controller.Speed.ProportionalGain = 1.0;
	gServoPnPInterface.Parameters.AxisAndDrivePars.Drive.Controller.Speed.IntegralTime = 0.0;
	gServoPnPInterface.Parameters.AxisAndDrivePars.Drive.Controller.Speed.FilterTime = 0.0;

	//these values are only used if controller mode is set to position + feed forward
	gServoPnPInterface.Parameters.AxisAndDrivePars.Drive.Controller.FeedForward.TorqueLoad = 0.0;
	gServoPnPInterface.Parameters.AxisAndDrivePars.Drive.Controller.FeedForward.TorquePositive = 0.0;
	gServoPnPInterface.Parameters.AxisAndDrivePars.Drive.Controller.FeedForward.TorqueNegative = 0.0;
	gServoPnPInterface.Parameters.AxisAndDrivePars.Drive.Controller.FeedForward.SpeedTorqueFactor = 0.0;
	gServoPnPInterface.Parameters.AxisAndDrivePars.Drive.Controller.FeedForward.Inertia = 0.0;
	gServoPnPInterface.Parameters.AxisAndDrivePars.Drive.Controller.FeedForward.AccelerationFilterTime = 0.0;
	gServoPnPInterface.Parameters.AxisAndDrivePars.Drive.DigitalInputs.Level.HomingSwitch = mpAXIS_IO_ACTIVE_HI_EXTERNAL;

	//feed

	strcpy((char*)&gServoFeedInterface.Parameters.AxisAndDrivePars.AxisName, "Feed");
	gServoFeedInterface.Parameters.AxisAndDrivePars.Axis.BaseType = mpAXIS_PERIODIC_LINEAR;
	gServoFeedInterface.Parameters.AxisAndDrivePars.Axis.MeasurementUnit = mpAXIS_UNIT_MM;
	gServoFeedInterface.Parameters.AxisAndDrivePars.Axis.MeasurementResolution = 0.01;
	gServoFeedInterface.Parameters.AxisAndDrivePars.Axis.SoftwareLimitPositions.LowerLimit = 0;
	gServoFeedInterface.Parameters.AxisAndDrivePars.Axis.SoftwareLimitPositions.UpperLimit = 360.0;
	gServoFeedInterface.Parameters.AxisAndDrivePars.Axis.PeriodSettings.Period = 711.2;

	gServoFeedInterface.Parameters.AxisAndDrivePars.Axis.MovementLimits.VelocityPositive = 1000.0;
	gServoFeedInterface.Parameters.AxisAndDrivePars.Axis.MovementLimits.VelocityNegative = 1000.0;
	gServoFeedInterface.Parameters.AxisAndDrivePars.Axis.MovementLimits.Acceleration = 10000.0;
	gServoFeedInterface.Parameters.AxisAndDrivePars.Axis.MovementLimits.Deceleration = 10000.0;
	gServoFeedInterface.Parameters.AxisAndDrivePars.Axis.MovementLimits.JerkTime = 0.0;
	gServoFeedInterface.Parameters.AxisAndDrivePars.Axis.MovementLimits.PositionErrorStopLimit = 2;
	gServoFeedInterface.Parameters.AxisAndDrivePars.Axis.MovementLimits.VelocityErrorStopLimit = 0.0;
	gServoFeedInterface.Parameters.AxisAndDrivePars.Axis.MovementLimits.VelocityErrorStopLimitMode = mpAXIS_VEL_MODE_OFF;

	//gServoFeedInterface.Parameters.AxisAndDrivePars.Axis.CyclicReadChannels.UserChannelParameterID = 214;

	gServoFeedInterface.Parameters.AxisAndDrivePars.Drive.Gearbox.Input = 10;
	gServoFeedInterface.Parameters.AxisAndDrivePars.Drive.Gearbox.Output = 1;
	gServoFeedInterface.Parameters.AxisAndDrivePars.Drive.Gearbox.Direction = mpAXIS_DIR_CLOCKWISE; //mpAXIS_DIR_CLOCKWISE is the normal rotation

	gServoFeedInterface.Parameters.AxisAndDrivePars.Drive.Transformation.ReferenceDistance = 279.4;

	//gServoFeedInterface.Parameters.AxisAndDrivePars.Drive.Controller.Mode = mpAXIS_CTRL_MODE_POSITION_FF;
	gServoFeedInterface.Parameters.AxisAndDrivePars.Drive.Controller.Mode = mpAXIS_CTRL_MODE_POSITION;
	gServoFeedInterface.Parameters.AxisAndDrivePars.Drive.Controller.Position.ProportionalGain = 400.0;
	gServoFeedInterface.Parameters.AxisAndDrivePars.Drive.Controller.Position.IntegralTime = 0.0;
	gServoFeedInterface.Parameters.AxisAndDrivePars.Drive.Controller.Position.PredictionTime = 0.0004;
	gServoFeedInterface.Parameters.AxisAndDrivePars.Drive.Controller.Position.TotalDelayTime = 0.0004;

	gServoFeedInterface.Parameters.AxisAndDrivePars.Drive.Controller.Speed.ProportionalGain = 0.6;
	gServoFeedInterface.Parameters.AxisAndDrivePars.Drive.Controller.Speed.IntegralTime = 0.1;
	gServoFeedInterface.Parameters.AxisAndDrivePars.Drive.Controller.Speed.FilterTime = 0.0;

	//these values are only used if controller mode is set to position + feed forward
	gServoFeedInterface.Parameters.AxisAndDrivePars.Drive.Controller.FeedForward.TorqueLoad = 0.0;
	gServoFeedInterface.Parameters.AxisAndDrivePars.Drive.Controller.FeedForward.TorquePositive = 0.0;
	gServoFeedInterface.Parameters.AxisAndDrivePars.Drive.Controller.FeedForward.TorqueNegative = 0.0;
	gServoFeedInterface.Parameters.AxisAndDrivePars.Drive.Controller.FeedForward.SpeedTorqueFactor = 0.0;
	gServoFeedInterface.Parameters.AxisAndDrivePars.Drive.Controller.FeedForward.Inertia = 0.0;
	gServoFeedInterface.Parameters.AxisAndDrivePars.Drive.Controller.FeedForward.AccelerationFilterTime = 0.0;

	// body hopper

	strcpy((char*)&gBodyHopperInterface.Parameters.AxisAndDrivePars.AxisName, "BodyHopper");
	gBodyHopperInterface.Parameters.AxisAndDrivePars.Axis.BaseType = mpAXIS_LINEAR;
	gBodyHopperInterface.Parameters.AxisAndDrivePars.Axis.MeasurementUnit = mpAXIS_UNIT_MM;
	gBodyHopperInterface.Parameters.AxisAndDrivePars.Axis.MeasurementResolution = 0.01;
	gBodyHopperInterface.Parameters.AxisAndDrivePars.Axis.SoftwareLimitPositions.LowerLimit = 0;
	gBodyHopperInterface.Parameters.AxisAndDrivePars.Axis.SoftwareLimitPositions.UpperLimit = 100.0;
	gBodyHopperInterface.Parameters.AxisAndDrivePars.Axis.PeriodSettings.Period = 360;

	gBodyHopperInterface.Parameters.AxisAndDrivePars.Axis.MovementLimits.VelocityPositive = 1000.0;
	gBodyHopperInterface.Parameters.AxisAndDrivePars.Axis.MovementLimits.VelocityNegative = 1000.0;
	gBodyHopperInterface.Parameters.AxisAndDrivePars.Axis.MovementLimits.Acceleration = 5000.0;
	gBodyHopperInterface.Parameters.AxisAndDrivePars.Axis.MovementLimits.Deceleration = 5000.0;
	gBodyHopperInterface.Parameters.AxisAndDrivePars.Axis.MovementLimits.JerkTime = 0.0;
	gBodyHopperInterface.Parameters.AxisAndDrivePars.Axis.MovementLimits.PositionErrorStopLimit = 2;
	gBodyHopperInterface.Parameters.AxisAndDrivePars.Axis.MovementLimits.VelocityErrorStopLimit = 0.0;
	gBodyHopperInterface.Parameters.AxisAndDrivePars.Axis.MovementLimits.VelocityErrorStopLimitMode = mpAXIS_VEL_MODE_OFF;

	//gBodyHopperInterface.Parameters.AxisAndDrivePars.Axis.CyclicReadChannels.UserChannelParameterID = 214;

	gBodyHopperInterface.Parameters.AxisAndDrivePars.Drive.Gearbox.Input = 10;
	gBodyHopperInterface.Parameters.AxisAndDrivePars.Drive.Gearbox.Output = 1;
	gBodyHopperInterface.Parameters.AxisAndDrivePars.Drive.Gearbox.Direction = mpAXIS_DIR_CLOCKWISE;

	gBodyHopperInterface.Parameters.AxisAndDrivePars.Drive.Transformation.ReferenceDistance = 381;

	//gBodyHopperInterface.Parameters.AxisAndDrivePars.Drive.Controller.Mode = mpAXIS_CTRL_MODE_POSITION_FF;
	gBodyHopperInterface.Parameters.AxisAndDrivePars.Drive.Controller.Mode = mpAXIS_CTRL_MODE_POSITION;
	gBodyHopperInterface.Parameters.AxisAndDrivePars.Drive.Controller.Position.ProportionalGain = 400.0;
	gBodyHopperInterface.Parameters.AxisAndDrivePars.Drive.Controller.Position.IntegralTime = 0.0;
	gBodyHopperInterface.Parameters.AxisAndDrivePars.Drive.Controller.Position.PredictionTime = 0.0004;
	gBodyHopperInterface.Parameters.AxisAndDrivePars.Drive.Controller.Position.TotalDelayTime = 0.0004;

	gBodyHopperInterface.Parameters.AxisAndDrivePars.Drive.Controller.Speed.ProportionalGain = 0.6;
	gBodyHopperInterface.Parameters.AxisAndDrivePars.Drive.Controller.Speed.IntegralTime = 0.1;
	gBodyHopperInterface.Parameters.AxisAndDrivePars.Drive.Controller.Speed.FilterTime = 0.0;

	//these values are only used if controller mode is set to position + feed forward
	gBodyHopperInterface.Parameters.AxisAndDrivePars.Drive.Controller.FeedForward.TorqueLoad = 0.0;
	gBodyHopperInterface.Parameters.AxisAndDrivePars.Drive.Controller.FeedForward.TorquePositive = 0.0;
	gBodyHopperInterface.Parameters.AxisAndDrivePars.Drive.Controller.FeedForward.TorqueNegative = 0.0;
	gBodyHopperInterface.Parameters.AxisAndDrivePars.Drive.Controller.FeedForward.SpeedTorqueFactor = 0.0;
	gBodyHopperInterface.Parameters.AxisAndDrivePars.Drive.Controller.FeedForward.Inertia = 0.0;
	gBodyHopperInterface.Parameters.AxisAndDrivePars.Drive.Controller.FeedForward.AccelerationFilterTime = 0.0;

	// left hopper

	strcpy((char*)&gLeftHopperInterface.Parameters.AxisAndDrivePars.AxisName, "LeftHopper");
	gLeftHopperInterface.Parameters.AxisAndDrivePars.Axis.BaseType = mpAXIS_LINEAR;
	gLeftHopperInterface.Parameters.AxisAndDrivePars.Axis.MeasurementUnit = mpAXIS_UNIT_MM;
	gLeftHopperInterface.Parameters.AxisAndDrivePars.Axis.MeasurementResolution = 0.01;
	gLeftHopperInterface.Parameters.AxisAndDrivePars.Axis.SoftwareLimitPositions.LowerLimit = 0;
	gLeftHopperInterface.Parameters.AxisAndDrivePars.Axis.SoftwareLimitPositions.UpperLimit = 100.0;
	gLeftHopperInterface.Parameters.AxisAndDrivePars.Axis.PeriodSettings.Period = 360;

	gLeftHopperInterface.Parameters.AxisAndDrivePars.Axis.MovementLimits.VelocityPositive = 1000.0;
	gLeftHopperInterface.Parameters.AxisAndDrivePars.Axis.MovementLimits.VelocityNegative = 1000.0;
	gLeftHopperInterface.Parameters.AxisAndDrivePars.Axis.MovementLimits.Acceleration = 5000.0;
	gLeftHopperInterface.Parameters.AxisAndDrivePars.Axis.MovementLimits.Deceleration = 5000.0;
	gLeftHopperInterface.Parameters.AxisAndDrivePars.Axis.MovementLimits.JerkTime = 0.0;
	gLeftHopperInterface.Parameters.AxisAndDrivePars.Axis.MovementLimits.PositionErrorStopLimit = 2;
	gLeftHopperInterface.Parameters.AxisAndDrivePars.Axis.MovementLimits.VelocityErrorStopLimit = 0.0;
	gLeftHopperInterface.Parameters.AxisAndDrivePars.Axis.MovementLimits.VelocityErrorStopLimitMode = mpAXIS_VEL_MODE_OFF;

	//gLeftHopperInterface.Parameters.AxisAndDrivePars.Axis.CyclicReadChannels.UserChannelParameterID = 214;

	gLeftHopperInterface.Parameters.AxisAndDrivePars.Drive.Gearbox.Input = 10;
	gLeftHopperInterface.Parameters.AxisAndDrivePars.Drive.Gearbox.Output = 1;
	gLeftHopperInterface.Parameters.AxisAndDrivePars.Drive.Gearbox.Direction = mpAXIS_DIR_COUNTERCLOCKWISE;

	gLeftHopperInterface.Parameters.AxisAndDrivePars.Drive.Transformation.ReferenceDistance = 381;

	//gLeftHopperInterface.Parameters.AxisAndDrivePars.Drive.Controller.Mode = mpAXIS_CTRL_MODE_POSITION_FF;
	gLeftHopperInterface.Parameters.AxisAndDrivePars.Drive.Controller.Mode = mpAXIS_CTRL_MODE_POSITION;
	gLeftHopperInterface.Parameters.AxisAndDrivePars.Drive.Controller.Position.ProportionalGain = 400.0;
	gLeftHopperInterface.Parameters.AxisAndDrivePars.Drive.Controller.Position.IntegralTime = 0.0;
	gLeftHopperInterface.Parameters.AxisAndDrivePars.Drive.Controller.Position.PredictionTime = 0.0004;
	gLeftHopperInterface.Parameters.AxisAndDrivePars.Drive.Controller.Position.TotalDelayTime = 0.0004;

	gLeftHopperInterface.Parameters.AxisAndDrivePars.Drive.Controller.Speed.ProportionalGain = 0.6;
	gLeftHopperInterface.Parameters.AxisAndDrivePars.Drive.Controller.Speed.IntegralTime = 0.1;
	gLeftHopperInterface.Parameters.AxisAndDrivePars.Drive.Controller.Speed.FilterTime = 0.0;

	//these values are only used if controller mode is set to position + feed forward
	gLeftHopperInterface.Parameters.AxisAndDrivePars.Drive.Controller.FeedForward.TorqueLoad = 0.0;
	gLeftHopperInterface.Parameters.AxisAndDrivePars.Drive.Controller.FeedForward.TorquePositive = 0.0;
	gLeftHopperInterface.Parameters.AxisAndDrivePars.Drive.Controller.FeedForward.TorqueNegative = 0.0;
	gLeftHopperInterface.Parameters.AxisAndDrivePars.Drive.Controller.FeedForward.SpeedTorqueFactor = 0.0;
	gLeftHopperInterface.Parameters.AxisAndDrivePars.Drive.Controller.FeedForward.Inertia = 0.0;
	gLeftHopperInterface.Parameters.AxisAndDrivePars.Drive.Controller.FeedForward.AccelerationFilterTime = 0.0;

	// right hopper

	strcpy((char*)&gRightHopperInterface.Parameters.AxisAndDrivePars.AxisName, "RightHopper");
	gRightHopperInterface.Parameters.AxisAndDrivePars.Axis.BaseType = mpAXIS_LINEAR;
	gRightHopperInterface.Parameters.AxisAndDrivePars.Axis.MeasurementUnit = mpAXIS_UNIT_MM;
	gRightHopperInterface.Parameters.AxisAndDrivePars.Axis.MeasurementResolution = 0.01;
	gRightHopperInterface.Parameters.AxisAndDrivePars.Axis.SoftwareLimitPositions.LowerLimit = 0;
	gRightHopperInterface.Parameters.AxisAndDrivePars.Axis.SoftwareLimitPositions.UpperLimit = 100.0;
	gRightHopperInterface.Parameters.AxisAndDrivePars.Axis.PeriodSettings.Period = 360;

	gRightHopperInterface.Parameters.AxisAndDrivePars.Axis.MovementLimits.VelocityPositive = 1000.0;
	gRightHopperInterface.Parameters.AxisAndDrivePars.Axis.MovementLimits.VelocityNegative = 1000.0;
	gRightHopperInterface.Parameters.AxisAndDrivePars.Axis.MovementLimits.Acceleration = 5000.0;
	gRightHopperInterface.Parameters.AxisAndDrivePars.Axis.MovementLimits.Deceleration = 5000.0;
	gRightHopperInterface.Parameters.AxisAndDrivePars.Axis.MovementLimits.JerkTime = 0.0;
	gRightHopperInterface.Parameters.AxisAndDrivePars.Axis.MovementLimits.PositionErrorStopLimit = 2;
	gRightHopperInterface.Parameters.AxisAndDrivePars.Axis.MovementLimits.VelocityErrorStopLimit = 0.0;
	gRightHopperInterface.Parameters.AxisAndDrivePars.Axis.MovementLimits.VelocityErrorStopLimitMode = mpAXIS_VEL_MODE_OFF;

	//gRightHopperInterface.Parameters.AxisAndDrivePars.Axis.CyclicReadChannels.UserChannelParameterID = 214;

	gRightHopperInterface.Parameters.AxisAndDrivePars.Drive.Gearbox.Input = 10;
	gRightHopperInterface.Parameters.AxisAndDrivePars.Drive.Gearbox.Output = 1;
	gRightHopperInterface.Parameters.AxisAndDrivePars.Drive.Gearbox.Direction = mpAXIS_DIR_COUNTERCLOCKWISE;

	gRightHopperInterface.Parameters.AxisAndDrivePars.Drive.Transformation.ReferenceDistance = 381;

	//gRightHopperInterface.Parameters.AxisAndDrivePars.Drive.Controller.Mode = mpAXIS_CTRL_MODE_POSITION_FF;
	gRightHopperInterface.Parameters.AxisAndDrivePars.Drive.Controller.Mode = mpAXIS_CTRL_MODE_POSITION;
	gRightHopperInterface.Parameters.AxisAndDrivePars.Drive.Controller.Position.ProportionalGain = 400.0;
	gRightHopperInterface.Parameters.AxisAndDrivePars.Drive.Controller.Position.IntegralTime = 0.0;
	gRightHopperInterface.Parameters.AxisAndDrivePars.Drive.Controller.Position.PredictionTime = 0.0004;
	gRightHopperInterface.Parameters.AxisAndDrivePars.Drive.Controller.Position.TotalDelayTime = 0.0004;

	gRightHopperInterface.Parameters.AxisAndDrivePars.Drive.Controller.Speed.ProportionalGain = 0.6;
	gRightHopperInterface.Parameters.AxisAndDrivePars.Drive.Controller.Speed.IntegralTime = 0.1;
	gRightHopperInterface.Parameters.AxisAndDrivePars.Drive.Controller.Speed.FilterTime = 0.0;

	//these values are only used if controller mode is set to position + feed forward
	gRightHopperInterface.Parameters.AxisAndDrivePars.Drive.Controller.FeedForward.TorqueLoad = 0.0;
	gRightHopperInterface.Parameters.AxisAndDrivePars.Drive.Controller.FeedForward.TorquePositive = 0.0;
	gRightHopperInterface.Parameters.AxisAndDrivePars.Drive.Controller.FeedForward.TorqueNegative = 0.0;
	gRightHopperInterface.Parameters.AxisAndDrivePars.Drive.Controller.FeedForward.SpeedTorqueFactor = 0.0;
	gRightHopperInterface.Parameters.AxisAndDrivePars.Drive.Controller.FeedForward.Inertia = 0.0;
	gRightHopperInterface.Parameters.AxisAndDrivePars.Drive.Controller.FeedForward.AccelerationFilterTime = 0.0;

	//******* End Axis and Drive Param Default Settings *******//

}

void _CYCLIC ProgramCyclic(void)
{

	//******************START RAM HANDLER******************//
	gIsSimulated = DiagCpuIsSimulated();

	if ((ServoRamFirstHomeExecuted == 0) || (ServoPnPFirstHomeExecuted == 0)) {
		gHMI.StatusDatapoints.ServoRamHomeSDP = UNHIDE;
	} else {
		gHMI.StatusDatapoints.ServoRamHomeSDP = HIDE;
	}

	gServoRamInterface.Commands.RequestHome = gHMI.Commands.HomeServoRam || ServoRamAutoHome;
	gServoRamInterface.Commands.RequestJogPos = gHMI.Commands.JogServoRamPos;
	gServoRamInterface.Commands.RequestJogNeg = gHMI.Commands.JogServoRamNeg;
	gServoRamInterface.Parameters.MovementParameters.Jog.Acceleration = gHMI.Parameters.ServoRamAccel;
	gServoRamInterface.Parameters.MovementParameters.Jog.Deceleration = gHMI.Parameters.ServoRamAccel;
	gServoRamInterface.Parameters.MovementParameters.Jog.Velocity = gHMI.Parameters.ServoRamJogVelocity;

	gServoRamInterface.Parameters.MovementParameters.Acceleration = gHMI.Parameters.ServoRamAccel;
	gServoRamInterface.Parameters.MovementParameters.Deceleration = gHMI.Parameters.ServoRamAccel;
	gServoRamInterface.Parameters.MovementParameters.Torque.Limit = gHMI.Parameters.ServoRamTorqueLimit;
	gServoRamInterface.Parameters.MovementParameters.CyclicRead.TorqueMode = mpAXIS_READ_CYCLIC;

	//update torque limit anytime it is changed
	if (gServoRamInterface.Status.AxisInitialized) {
		if (OldTorqueLimitRam != gServoRamInterface.Parameters.MovementParameters.Torque.Limit) {
			gServoRamInterface.Commands.ToMapp.Update = 1;
		}

		OldTorqueLimitRam = gServoRamInterface.Parameters.MovementParameters.Torque.Limit;
	}

	//home request while running should clear command to cycle the ram This prevents ram from taking off immediately after home complets
	if (gServoRamInterface.Commands.RequestHome) {
		gHMI.Commands.CycleServoRam = 0;
	}

	//OldTorqueLimitRam = gServoRamInterface.Parameters.MovementParameters.Torque.Limit;

	ServoRamHandler.AlarmActive = gHighSeverityAlarmActive;
	ServoRamHandler.IsSimulated = gIsSimulated;
	ServoRamHandler.FirstHomeExecuted = &ServoRamFirstHomeExecuted;
	ServoRamHandler.pInterface = &gServoRamInterface;
	ServoRamHandler.pHomingParameters = &gHomingParameters.ServoRam;
	AxisHandler(&ServoRamHandler);;
	//******************END RAM HANDLER******************//

	//******************START FEED HANDLER******************//
	gServoFeedInterface.Commands.RequestHome = gHMI.Commands.HomeServoFeed;
	gServoFeedInterface.Commands.RequestJogPos = gHMI.Commands.JogServoFeedPos;
	gServoFeedInterface.Commands.RequestJogNeg = gHMI.Commands.JogServoFeedNeg;
	gServoFeedInterface.Parameters.MovementParameters.Jog.Acceleration = gHMI.Parameters.ServoFeedAccel;
	gServoFeedInterface.Parameters.MovementParameters.Jog.Deceleration = gHMI.Parameters.ServoFeedAccel;
	gServoFeedInterface.Parameters.MovementParameters.Jog.Velocity = gHMI.Parameters.ServoFeedJogVelocity;

	gServoFeedInterface.Parameters.MovementParameters.Acceleration = gHMI.Parameters.ServoFeedAccel;
	gServoFeedInterface.Parameters.MovementParameters.Deceleration = gHMI.Parameters.ServoFeedAccel;
	gServoFeedInterface.Parameters.MovementParameters.Velocity = gHMI.Parameters.ServoFeedVelocity;
	gServoFeedInterface.Parameters.MovementParameters.Torque.Limit = gHMI.Parameters.ServoFeedTorqueLimit;

	//update torque limit anytime it is changed
	if (gServoFeedInterface.Status.AxisInitialized) {
		if (OldTorqueLimitFeed != gServoFeedInterface.Parameters.MovementParameters.Torque.Limit) {
			gServoFeedInterface.Commands.ToMapp.Update = 1;
		}

		OldTorqueLimitFeed = gServoFeedInterface.Parameters.MovementParameters.Torque.Limit;
	}

	ServoFeedHandler.AlarmActive = gHighSeverityAlarmActive;
	ServoFeedHandler.IsSimulated = gIsSimulated;
	ServoFeedHandler.FirstHomeExecuted = &ServoFeedFirstHomeExecuted;
	ServoFeedHandler.pInterface = &gServoFeedInterface;
	ServoFeedHandler.pHomingParameters = &gHomingParameters.ServoFeed;
	AxisHandler(&ServoFeedHandler);
	//******************END FEED HANDLER******************//

	//******************START BODY HOPPER HANDLER******************//
	gBodyHopperInterface.Commands.RequestHome = gHMI.Commands.HomeBodyHopper;
	gBodyHopperInterface.Commands.RequestJogPos = gHMI.Commands.JogBodyHopperPos;
	gBodyHopperInterface.Commands.RequestJogNeg = gHMI.Commands.JogBodyHopperNeg;
	gBodyHopperInterface.Parameters.MovementParameters.Jog.Acceleration = gHMI.Parameters.BodyHopperAccel;
	gBodyHopperInterface.Parameters.MovementParameters.Jog.Deceleration = gHMI.Parameters.BodyHopperAccel;
	gBodyHopperInterface.Parameters.MovementParameters.Jog.Velocity = gHMI.Parameters.BodyHopperJogVelocity;

	gBodyHopperInterface.Parameters.MovementParameters.Acceleration = gHMI.Parameters.BodyHopperAccel;
	gBodyHopperInterface.Parameters.MovementParameters.Deceleration = gHMI.Parameters.BodyHopperAccel;
	gBodyHopperInterface.Parameters.MovementParameters.Velocity = gHMI.Parameters.BodyHopperVelocity;
	gBodyHopperInterface.Parameters.MovementParameters.Torque.Limit = gHMI.Parameters.BodyHopperTorqueLimit;
	gBodyHopperInterface.Parameters.MovementParameters.CyclicRead.TorqueMode = mpAXIS_READ_CYCLIC;

	//update torque limit anytime it is changed
	if (gBodyHopperInterface.Status.AxisInitialized) {
		if (OldTorqueLimitBodyHopper != gBodyHopperInterface.Parameters.MovementParameters.Torque.Limit) {
			gBodyHopperInterface.Commands.ToMapp.Update = 1;
		}

		OldTorqueLimitBodyHopper = gBodyHopperInterface.Parameters.MovementParameters.Torque.Limit;
	}

	BodyHopperHandler.AlarmActive = gHighSeverityAlarmActive;
	BodyHopperHandler.IsSimulated = gIsSimulated;
	BodyHopperHandler.FirstHomeExecuted = &BodyHopperFirstHomeExecuted;
	BodyHopperHandler.pInterface = &gBodyHopperInterface;
	BodyHopperHandler.pHomingParameters = &gHomingParameters.BodyHopper;
	AxisHandler(&BodyHopperHandler);
	//******************END BODY HOPPER HANDLER******************//

	//******************START LEFT HOPPER HANDLER******************//
	gBodyHopperInterface.Commands.RequestHome = gHMI.Commands.HomeBodyHopper;
	gLeftHopperInterface.Commands.RequestJogPos = gHMI.Commands.JogLeftHopperPos;
	gLeftHopperInterface.Commands.RequestJogNeg = gHMI.Commands.JogLeftHopperNeg;
	gLeftHopperInterface.Parameters.MovementParameters.Jog.Acceleration = gHMI.Parameters.LeftHopperAccel;
	gLeftHopperInterface.Parameters.MovementParameters.Jog.Deceleration = gHMI.Parameters.LeftHopperAccel;
	gLeftHopperInterface.Parameters.MovementParameters.Jog.Velocity = gHMI.Parameters.LeftHopperJogVelocity;

	gLeftHopperInterface.Parameters.MovementParameters.Acceleration = gHMI.Parameters.LeftHopperAccel;
	gLeftHopperInterface.Parameters.MovementParameters.Deceleration = gHMI.Parameters.LeftHopperAccel;
	gLeftHopperInterface.Parameters.MovementParameters.Velocity = gHMI.Parameters.LeftHopperVelocity;
	gLeftHopperInterface.Parameters.MovementParameters.Torque.Limit = gHMI.Parameters.LeftHopperTorqueLimit;
	gLeftHopperInterface.Parameters.MovementParameters.CyclicRead.TorqueMode = mpAXIS_READ_CYCLIC;

	//update torque limit anytime it is changed
	if (gLeftHopperInterface.Status.AxisInitialized) {
		if (OldTorqueLimitLeftHopper != gLeftHopperInterface.Parameters.MovementParameters.Torque.Limit) {
			gLeftHopperInterface.Commands.ToMapp.Update = 1;
		}

		OldTorqueLimitLeftHopper = gLeftHopperInterface.Parameters.MovementParameters.Torque.Limit;
	}

	LeftHopperHandler.AlarmActive = gHighSeverityAlarmActive;
	LeftHopperHandler.IsSimulated = gIsSimulated;
	LeftHopperHandler.FirstHomeExecuted = &LeftHopperFirstHomeExecuted;
	LeftHopperHandler.pInterface = &gLeftHopperInterface;
	LeftHopperHandler.pHomingParameters = &gHomingParameters.LeftHopper;
	AxisHandler(&LeftHopperHandler);
	//******************END LEFT HOPPER HANDLER******************//

	//******************START RIGHT HOPPER HANDLER******************//
	gBodyHopperInterface.Commands.RequestHome = gHMI.Commands.HomeRightHopper;
	gRightHopperInterface.Commands.RequestJogPos = gHMI.Commands.JogRightHopperPos;
	gRightHopperInterface.Commands.RequestJogNeg = gHMI.Commands.JogRightHopperNeg;
	gRightHopperInterface.Parameters.MovementParameters.Jog.Acceleration = gHMI.Parameters.RightHopperAccel;
	gRightHopperInterface.Parameters.MovementParameters.Jog.Deceleration = gHMI.Parameters.RightHopperAccel;
	gRightHopperInterface.Parameters.MovementParameters.Jog.Velocity = gHMI.Parameters.RightHopperJogVelocity;

	gRightHopperInterface.Parameters.MovementParameters.Acceleration = gHMI.Parameters.RightHopperAccel;
	gRightHopperInterface.Parameters.MovementParameters.Deceleration = gHMI.Parameters.RightHopperAccel;
	gRightHopperInterface.Parameters.MovementParameters.Velocity = gHMI.Parameters.RightHopperVelocity;
	gRightHopperInterface.Parameters.MovementParameters.Torque.Limit = gHMI.Parameters.RightHopperTorqueLimit;
	gRightHopperInterface.Parameters.MovementParameters.CyclicRead.TorqueMode = mpAXIS_READ_CYCLIC;

	//update torque limit anytime it is changed
	if (gRightHopperInterface.Status.AxisInitialized) {
		if (OldTorqueLimitRightHopper != gRightHopperInterface.Parameters.MovementParameters.Torque.Limit) {
			gRightHopperInterface.Commands.ToMapp.Update = 1;
		}

		OldTorqueLimitRightHopper = gRightHopperInterface.Parameters.MovementParameters.Torque.Limit;
	}

	RightHopperHandler.AlarmActive = gHighSeverityAlarmActive;
	RightHopperHandler.IsSimulated = gIsSimulated;
	RightHopperHandler.FirstHomeExecuted = &RightHopperFirstHomeExecuted;
	RightHopperHandler.pInterface = &gRightHopperInterface;
	RightHopperHandler.pHomingParameters = &gHomingParameters.RightHopper;
	AxisHandler(&RightHopperHandler);
	//******************END RIGHT HOPPER HANDLER******************//

		//******************START PNP HANDLER******************//
	gServoPnPInterface.Commands.RequestHome = gHMI.Commands.HomeServoPnP || ServoPnPAutoHome;
	gServoPnPInterface.Commands.RequestJogPos = gHMI.Commands.JogServoPnPPos;
	gServoPnPInterface.Commands.RequestJogNeg = gHMI.Commands.JogServoPnPNeg;
	gServoPnPInterface.Parameters.MovementParameters.Jog.Acceleration = gHMI.Parameters.ServoPnPAccel;
	gServoPnPInterface.Parameters.MovementParameters.Jog.Deceleration = gHMI.Parameters.ServoPnPAccel;
	gServoPnPInterface.Parameters.MovementParameters.Jog.Velocity = gHMI.Parameters.ServoPnPJogVelocity;

	gServoPnPInterface.Parameters.MovementParameters.Acceleration = gHMI.Parameters.ServoPnPAccel;
	gServoPnPInterface.Parameters.MovementParameters.Deceleration = gHMI.Parameters.ServoPnPAccel;
	gServoPnPInterface.Parameters.MovementParameters.Torque.Limit = gHMI.Parameters.ServoPnPTorqueLimit;
	gServoPnPInterface.Parameters.MovementParameters.CyclicRead.TorqueMode = mpAXIS_READ_CYCLIC;

	//update torque limit anytime it is changed
	if (gServoPnPInterface.Status.AxisInitialized) {
		if (OldTorqueLimitRam != gServoPnPInterface.Parameters.MovementParameters.Torque.Limit) {
			gServoPnPInterface.Commands.ToMapp.Update = 1;
		}

		OldTorqueLimitRam = gServoPnPInterface.Parameters.MovementParameters.Torque.Limit;
	}

	//home request while running should clear command to cycle the ram This prevents ram from taking off immediately after home complets
	if (gServoPnPInterface.Commands.RequestHome) {
		gHMI.Commands.CycleServoPnP = 0;
	}

	//OldTorqueLimitRam = gServoPnPInterface.Parameters.MovementParameters.Torque.Limit;

	ServoPnPHandler.AlarmActive = gHighSeverityAlarmActive;
	ServoPnPHandler.IsSimulated = gIsSimulated;
	ServoPnPHandler.FirstHomeExecuted = &ServoPnPFirstHomeExecuted;
	ServoPnPHandler.pInterface = &gServoPnPInterface;
	ServoPnPHandler.pHomingParameters = &gHomingParameters.ServoPnP;
	AxisHandler(&ServoPnPHandler);
	//******************END PNP HANDLER******************//

	// Call FUBS
	SetHardwareInputs.HomeSwitch = gIO.DIs.BodyPickHome;
	SetHardwareInputs.Axis = &gServoPnP;
	SetHardwareInputs.Enable = 1;
	MC_BR_SetHardwareInputs(&SetHardwareInputs);
}

void _EXIT ProgramExit(void)
{

}
```

### Program Logical/ServoMotion/ServoPnPHandler

#### Main.st
```iecst
PROGRAM _INIT

	// Velocities and Accels
	gHMI.Parameters.ServoPnPJogVelocity := 10;
	gHMI.Parameters.ServoPnPPositiveVelocity := 90.0;
	gHMI.Parameters.ServoPnPNegativeVelocity := 90.0;
	gHMI.Parameters.ServoPnPAccel := 1000.0;

	// Positions
	gHMI.Parameters.ServoPnPStartPosition := 0;
	gHMI.Parameters.ServoPnPVacuumOffPosition := 80; //this is the position where the vacuum will be turned off on the way down to horizontal
	gHMI.Parameters.ServoPnPEndPosition := 110;
	//105 was the original position. Found that the box was rubbing the suction cups.

	// Times
	gHMI.Parameters.ServoPnPStartDwellTime := 100;
	gHMI.Parameters.BodyKickerTime := 250;
	gHMI.Parameters.BodyKickerRetractTime := 500;

	// Other
	gHMI.Parameters.ServoPnPTorqueLimit := 3.0;	//3 is original setting.

END_PROGRAM

PROGRAM _CYCLIC

	IF gHighSeverityAlarmActive THEN
		state := SERVOPNP_ERROR;
	END_IF

	StartDwellTimer.IN := FALSE; //Set in state machine if needed
	BodyKickerTimer.IN := FALSE;
	BodyKickerRetractTimer.IN := FALSE;

//	IF (NOT gHMI.Commands.CycleServoPnP AND NOT SingleCyclePnP) AND state <> SERVOPNP_ERROR AND gServoPnPInterface.Status.Homed THEN
//		state := SERVOPNP_IDLE;
//	END_IF

	// Resetting clears the grab alarm
	IF gHMI.Commands.RequestReset THEN
		BodyGrabFailAlarm := FALSE;
	END_IF

	CASE state OF

		SERVOPNP_WAIT_FOR_HOME:

            // Pick and place should home automatically on machine start up.
			IF gServoPnPInterface.Status.Homed AND ServoPnPFirstHomeExecuted THEN
				ServoPnPAutoHome := FALSE;
				gPnPAtStopPosition := TRUE;
				gHMI.Commands.CycleServoPnP := FALSE;
				gServoPnPInterface.Commands.ToMapp.TorqueLimitingOn := TRUE; //turn torque limiting on
				state := SERVOPNP_IDLE;
			ELSIF gServoPnPInterface.Status.PoweredOn AND NOT ServoPnPFirstHomeExecuted THEN
                ServoPnPAutoHome := TRUE;
                //GuideCylinder    := FALSE;
				state := SERVOPNP_WAIT_FOR_AUTO_HOME;
			END_IF

		SERVOPNP_WAIT_FOR_AUTO_HOME:

			IF gServoPnPInterface.Status.Homed AND ServoPnPFirstHomeExecuted THEN
				ServoPnPAutoHome := FALSE;
				gPnPAtStopPosition := TRUE;
				gHMI.Commands.CycleServoPnP := FALSE;
				gServoPnPInterface.Commands.ToMapp.TorqueLimitingOn := TRUE; //turn torque limiting on
				state := SERVOPNP_IDLE;
			END_IF

		SERVOPNP_IDLE:

			ServoPnPAutoHome := FALSE;
			gServoPnPInterface.Status.MoveComplete := FALSE;

            // Wait for the run command, then go to the start position
			IF (gHMI.Commands.CycleServoPnP OR (SingleCyclePnP)) AND ServoPnPFirstHomeExecuted THEN
				gCyclesToFinish := gCyclesToFinish + 1;
				gServoPnPInterface.Parameters.MovementParameters.Position := gHMI.Parameters.ServoPnPStartPosition;
				gServoPnPInterface.Parameters.MovementParameters.Velocity := gHMI.Parameters.ServoPnPPositiveVelocity;
				gServoPnPInterface.Commands.RequestMoveAbs := TRUE;
				state := SERVOPNP_MOVE_TO_HOPPER;
			END_IF

		SERVOPNP_MOVE_TO_HOPPER:

            GuideCylinder    := FALSE;

			// At the hopper position, if the body hopper is on, turn on the vacuum and dwell if there is a dwell time, or move to horizontal
			IF gServoPnPInterface.Status.MoveComplete AND gIO.DIs.BodyHopperMotor_RUN THEN
				gIO.DOs.BodyVacuumOn := TRUE;
				gServoPnPInterface.Status.MoveComplete := FALSE;
				IF gHMI.Parameters.ServoPnPStartDwellTime > 0 THEN
					state := SERVOPNP_DWELL_AT_HOPPER;
				ELSE
					gServoPnPInterface.Parameters.MovementParameters.Position := gHMI.Parameters.ServoPnPEndPosition;
					gServoPnPInterface.Parameters.MovementParameters.Velocity := gHMI.Parameters.ServoPnPNegativeVelocity;
					gServoPnPInterface.Commands.RequestMoveAbs := TRUE;
					state := SERVOPNP_MOVE_TO_HORIZONTAL;
				END_IF
			END_IF

		SERVOPNP_DWELL_AT_HOPPER:

            // Wait for the timer to finish, then start the move towards horizontal
            StartDwellTimer.IN := TRUE;
			IF StartDwellTimer.Q THEN
				StartDwellTimer.IN := FALSE;
				gServoPnPInterface.Parameters.MovementParameters.Position := gHMI.Parameters.ServoPnPEndPosition;
				gServoPnPInterface.Parameters.MovementParameters.Velocity := gHMI.Parameters.ServoPnPNegativeVelocity;
				gServoPnPInterface.Commands.RequestMoveAbs := TRUE;
				state := SERVOPNP_CHECK_FOR_BOX;
			END_IF

		SERVOPNP_CHECK_FOR_BOX:

			// After rotating 20 degrees, check that a box is actually grabbed
			IF gServoPnPInterface.Status.ActualPosition > 20 THEN
				IF gIO.DIs.BodyVacuumAchieved THEN
					// If the vacuum was achieved, then continue the move to horizontal
					FailureCount := 0;
					state := SERVOPNP_MOVE_TO_HORIZONTAL;
				ELSE
					FailureCount := FailureCount + 1;
					// If the vacuum failed, a box was not grabbed. Unless this was the third failure, try again
					IF FailureCount = NUM_PNP_TRIES THEN
						BodyGrabFailAlarm := TRUE;
						// Return home
						gServoPnPInterface.Parameters.MovementParameters.Position := gHMI.Parameters.ServoPnPStartPosition;
						gServoPnPInterface.Parameters.MovementParameters.Velocity := gHMI.Parameters.ServoPnPPositiveVelocity;
						gServoPnPInterface.Commands.RequestMoveAbs := TRUE;
						state := SERVOPNP_ERROR;
                    ELSE
						state := SERVOPNP_ABORT_AND_RETURN;
					END_IF
				END_IF
			END_IF

		SERVOPNP_MOVE_TO_HORIZONTAL:

			IF gServoPnPInterface.Status.ActualPosition > gHMI.Parameters.ServoPnPVacuumOffPosition THEN
				gIO.DOs.BodyVacuumOn := FALSE;
			END_IF

			// At the horizontal position, cut off the vacuum
			IF gServoPnPInterface.Status.MoveComplete THEN
				gIO.DOs.BodyVacuumOn := FALSE;
				// Wait for the ram to be ready (sucessful side folds) then push the box to the feeder and wait for it to clear
				IF (SingleCyclePnP) THEN
					SingleCyclePnP := FALSE;
					state := SERVOPNP_IDLE;
				ELSIF (*gIO.DIs.SideFoldVacuumAchieved AND *) gServoRamInterface.Status.ClearOfRoller AND gRamWaitingOnBox THEN
					gServoPnPInterface.Status.MoveComplete := FALSE;
					gIO.DOs.BodyKicker := TRUE;
					state := SERVOPNP_REMOVE_BOX;
				END_IF
			END_IF

        SERVOPNP_REMOVE_BOX:

            GuideCylinder := TRUE;
			// After the delay, turn off the kicker and start the retract timer
			BodyKickerTimer.IN := TRUE;
			IF BodyKickerTimer.Q THEN
				gIO.DOs.BodyKicker := FALSE;
				BodyKickerRetractTimer.IN := TRUE;
			END_IF
			// When the retract timer is done and the adhesive photoeye falls, send the pick and place home
			FTrig_AdhesivePhotoeye(CLK:=gIO.DIs.AdhesivePhotoEye);
			IF FTrig_AdhesivePhotoeye.Q AND BodyKickerRetractTimer.Q THEN
				BodyKickerTimer.IN := FALSE;
				BodyKickerRetractTimer.IN := FALSE;

				IF (NOT gHMI.Commands.CycleServoPnP) THEN
					state := SERVOPNP_IDLE;
				ELSE
					// On the falling edge of the adhesive photoeye, send the pick and place back to the hopper
					gCyclesToFinish := gCyclesToFinish + 1;
					gServoPnPInterface.Parameters.MovementParameters.Position := gHMI.Parameters.ServoPnPStartPosition;
					gServoPnPInterface.Parameters.MovementParameters.Velocity := gHMI.Parameters.ServoPnPPositiveVelocity;
                    gServoPnPInterface.Commands.RequestMoveAbs := TRUE;
                    //GuideCylinder := TRUE;
					state := SERVOPNP_MOVE_TO_HOPPER;
				END_IF
			END_IF

        SERVOPNP_ABORT_AND_RETURN:
            IF gServoPnPInterface.Status.MoveComplete THEN
                gServoPnPInterface.Status.MoveComplete := FALSE;
                gServoPnPInterface.Parameters.MovementParameters.Position := gHMI.Parameters.ServoPnPStartPosition;
                gServoPnPInterface.Parameters.MovementParameters.Velocity := gHMI.Parameters.ServoPnPNegativeVelocity;
                gServoPnPInterface.Commands.RequestMoveAbs := TRUE;
                state := SERVOPNP_MOVE_TO_HOPPER;
            END_IF

		SERVOPNP_ERROR:
            // Error response
			gServoPnPInterface.Status.MoveComplete := FALSE;
			gHMI.Commands.CycleServoPnP := FALSE;
			ServoPnPAutoHome := FALSE;
			gServoPnPInterface.Commands.RequestMoveAbs := FALSE;
			gIO.DOs.BodyVacuumOn := FALSE;
			gIO.DOs.BodyKicker := FALSE;
			SingleCyclePnP := FALSE;
			IF (gNumActiveAlarms = 0) THEN
				FailureCount := 0;
				state := SERVOPNP_WAIT_FOR_HOME;
			END_IF

	END_CASE;

	//The kicker is not allowed to be on if the servo PNP is below 97 degrees (Smaller number => further from horizontal)
	IF gServoPnPInterface.Status.ActualPosition < 97.0 THEN
		gIO.DOs.BodyKicker := FALSE;
	END_IF

	StartDwellTimer.PT := gHMI.Parameters.ServoPnPStartDwellTime;
	StartDwellTimer();
	BodyKickerTimer.PT := gHMI.Parameters.BodyKickerTime;
	BodyKickerTimer();
	BodyKickerRetractTimer.PT := gHMI.Parameters.BodyKickerRetractTime;
    BodyKickerRetractTimer();

//    IF gForceBodyKicker THEN
//        gIO.DOs.BodyKicker := TRUE;
//    ELSE
//        gIO.DOs.BodyKicker := FALSE;
//    END_IF

	END_PROGRAM

PROGRAM _EXIT
				(* Insert code here *)

				END_PROGRAM
```

### Program Logical/ServoMotion/ServoRamHandler

#### Main.st
```iecst
PROGRAM _INIT

	// Velocities and Accels
	gHMI.Parameters.ServoRamJogVelocity := 50;

	gHMI.Parameters.ServoRamSideFormingVelocity := 500.0;
	gHMI.Parameters.ServoRamBoxFormingVelocity := 750.0;
	gHMI.Parameters.ServoRamNegativeVelocity := 750.0;

	gHMI.Parameters.ServoRamAccel := 2000.0; //values much higher than this create an audible pop sound as tension changes direction in the belt at end of travel

	// Positions
	gHMI.Parameters.ServoRamStartPosition := 14.72;
	gHMI.Parameters.ServoRamMiddlePosition := 255.0;
	gHMI.Parameters.ServoRamFoldStartPos := 75.0;
	gHMI.Parameters.ServoRamFoldEndPos := 290.0;
	gHMI.Parameters.ServoRamEndPosition := 805.0;

	// Times
	gHMI.Parameters.ServoRamEndDwellTime := 100;
	gHMI.Parameters.ServoRamStartDwellTime := 100;
	gHMI.Parameters.ServoRamSidePickTime:= 300;
	gHMI.Parameters.ServoRamSidePickRetractTime := 300;
	gHMI.Parameters.ServoRamSideFoldTime:= 100;
	gHMI.Parameters.ServoRamSideFoldRetractTime := 50;
	gHMI.Parameters.RamDelay := 100;

	// Other
	gHMI.Parameters.ServoRamTorqueLimit := 6.0;
	gHMI.Parameters.ServoRamClearPosition := 300;

	//	gHMI.Parameters.ServoRamTimeoutTime := T#3s;

	gPassword; //need to use this somewhere. Was getting thrown out in slimmed down test code for servo ram

END_PROGRAM

PROGRAM _CYCLIC

	IF gHighSeverityAlarmActive THEN
		state := SERVORAM_ERROR;
	END_IF

	gIO.DOs.ResetSafety := gHMI.Commands.RequestReset OR ForceSafetyReset;

	// Resetting clears the grab and fold alarms
	IF gHMI.Commands.RequestReset THEN
		SideGrabFailAlarm := FALSE;
		SideFoldFailAlarm := FALSE;
		ResetTimeoutAlarm := FALSE;
	END_IF

	// Automatically disable all timers. Explicitly set them in state machine when needed
	EndDwellTimer.IN := FALSE;
	SidePickTimer.IN := FALSE;
	SidePickRetractTimer.IN := FALSE;
	SideFoldTimer.IN := FALSE;
	SideFoldRetractTimer.IN := FALSE;
	RamDelayTimer.IN := FALSE;
	ResetTimeoutTimer.IN := FALSE;

	// If the hopper has been reset but the machine isn't running, only let the hopper run for an alotted time to protect the motor
	IF NOT gHMI.Commands.CycleServoRam AND NOT gServoRamInterface.Status.Error THEN
		ResetTimeoutTimer.IN := TRUE;
	END_IF
	IF ResetTimeoutTimer.Q THEN
		//	ResetTimeoutAlarm := TRUE;
	END_IF

	IF gServoRamInterface.Status.ActualPosition <= gHMI.Parameters.ServoRamClearPosition THEN
		gServoRamInterface.Status.ClearOfRoller := TRUE;
	ELSE
		gServoRamInterface.Status.ClearOfRoller := FALSE;
	END_IF

//	IF NOT gHMI.Commands.CycleServoRam AND NOT ExerciseRam AND state <> SERVORAM_ERROR AND gServoRamInterface.Status.Homed THEN
//		state := SERVORAM_IDLE;
//	END_IF

	CASE state OF

		SERVORAM_WAIT_FOR_HOME:

			// Servo ram should home automatically on machine start up.
			IF gServoRamInterface.Status.Homed AND ServoRamFirstHomeExecuted THEN
				ServoRamAutoHome := FALSE;
				gRamAtStopPosition := TRUE;
				gHMI.Commands.CycleServoRam := FALSE;
				gServoRamInterface.Commands.ToMapp.TorqueLimitingOn := TRUE; //turn torque limiting on
				state := SERVORAM_IDLE;
			ELSIF gServoRamInterface.Status.PoweredOn AND NOT ServoRamFirstHomeExecuted THEN
				ServoRamAutoHome := TRUE;
				state := SERVORAM_WAIT_FOR_AUTO_HOME;
			END_IF

		SERVORAM_WAIT_FOR_AUTO_HOME:

			IF gServoRamInterface.Status.Homed AND ServoRamFirstHomeExecuted THEN
				ServoRamAutoHome := FALSE;
				gRamAtStopPosition := TRUE;
				gHMI.Commands.CycleServoRam := FALSE;
				gServoRamInterface.Commands.ToMapp.TorqueLimitingOn := TRUE; //turn torque limiting on
				state := SERVORAM_IDLE;
			END_IF

		SERVORAM_IDLE:

			ServoRamAutoHome := FALSE;
			gServoRamInterface.Status.MoveComplete := FALSE; //if we force a transition to IDLE while moving, we may have a stuck move complete flag. clear it here

			gCyclesToFinish := 0;

			// Wait for the ram to be homed and for run to be pressed, then move to the starting position
			IF gHMI.Commands.CycleServoRam AND ServoRamFirstHomeExecuted THEN
				ServoRamBusy := TRUE;
				gRamWaitingOnBox := TRUE; //tell the PnP that we are waiting on a box
				gServoRamInterface.Commands.ToMapp.TorqueLimitingOn := TRUE; //turn torque limiting on
				gServoRamInterface.Parameters.MovementParameters.Position := gHMI.Parameters.ServoRamStartPosition;
				gServoRamInterface.Parameters.MovementParameters.Velocity := gHMI.Parameters.ServoRamNegativeVelocity;
				gServoRamInterface.Commands.RequestMoveAbs := TRUE;
				gRamAtStopPosition := FALSE;
				ServoRamBusy := TRUE;
				state := SERVORAM_MOVE_TO_START;

				//allow the ram to cycle through the start, middle, and end positions. Lets us exercise the movements without using actuators
				//this should only be used to test the machine
			ELSIF ExerciseRam THEN
				gServoRamInterface.Commands.ToMapp.TorqueLimitingOn := TRUE; //turn torque limiting on
				gServoRamInterface.Parameters.MovementParameters.Position := gHMI.Parameters.ServoRamStartPosition;
				gServoRamInterface.Parameters.MovementParameters.Velocity := gHMI.Parameters.ServoRamNegativeVelocity;
				gServoRamInterface.Commands.RequestMoveAbs := TRUE;
				state := SERVORAM_MOVE_TO_START_EX;
			END_IF

		SERVORAM_MOVE_TO_START:

			// At the starting position, turn on the side vacuum and push the cylinders out to grab the side panels
			// The left and right hoppers must be on, the feed wheels must be running, and the PNP must have left its home position
			IF NOT gHMI.Commands.CycleServoRam AND gServoRamInterface.Status.MoveComplete AND (gCyclesToFinish = 0) THEN
				gServoRamInterface.Status.MoveComplete := FALSE;
				state := SERVORAM_IDLE;
			ELSIF gServoRamInterface.Status.MoveComplete AND gIO.DIs.LeftHopperMotor_RUN AND gIO.DIs.RightHopperMotor_RUN AND gIO.DIs.BodyHopperMotor_RUN AND
				gServoFeedInterface.Status.InMotion AND NOT gIO.DIs.BodyPickHome (*AND gIO.DIs.BodyVacuumAchieved*) AND (gCyclesToFinish > 0) THEN
				gRamAtStopPosition := TRUE;
				gServoRamInterface.Status.MoveComplete := FALSE;
				ServoRamBusy := FALSE;
				gIO.DOs.SidePanelVacOn := TRUE;
				gIO.DOs.SidePanelHoldVacuum := TRUE;
				gIO.DOs.SidePickCylinder := TRUE;
				state := SERVORAM_PICK_SIDES;
			END_IF

		SERVORAM_PICK_SIDES:
			SidePickTimer.IN := TRUE;
			// Wait for the side pick timer, then retract the side pick
			IF SidePickTimer.Q THEN
				gIO.DOs.SidePickCylinder := FALSE;
				SidePickRetractTimer.IN := TRUE;
			END_IF
			// When the side pick is retracted, check for side panels
			IF SidePickRetractTimer.Q THEN
				SidePickTimer.IN := FALSE;
				SidePickRetractTimer.IN := FALSE;
				state := SERVORAM_CHECK_FOR_SIDES;
			END_IF

		SERVORAM_CHECK_FOR_SIDES:
			IF gIO.DIs.SidePickVacuumAchieved THEN
				// If the side pick has vacuum, then the sides were picked, move to middle position
				SideFailureCount := 0;
				state := SERVORAM_WAITING_ON_BOX;
			ELSE
				// If vacuum was not achieved, then the side pick failed. Increment the fail counter
				SideFailureCount := SideFailureCount + 1;
				IF SideFailureCount = NUM_SIDE_TRIES THEN
					// If the side fails too many times, raise an error
					SideGrabFailAlarm := TRUE;
					state := SERVORAM_ERROR;
				ELSE
					// Otherwise, try again
					gIO.DOs.SidePickCylinder := TRUE;
					state := SERVORAM_PICK_SIDES;
				END_IF
			END_IF

		SERVORAM_WAITING_ON_BOX:
			// Run the delay timer when a box is seen
			RamDelayTimer.IN := gIO.DIs.BodyDetect;
			// When the delay finishes, move the ram to the end position
			IF gIO.DIs.SidePickVacuumAchieved AND RamDelayTimer.Q THEN
				gServoRamInterface.Parameters.MovementParameters.Position := gHMI.Parameters.ServoRamEndPosition;
				gServoRamInterface.Parameters.MovementParameters.Velocity := gHMI.Parameters.ServoRamBoxFormingVelocity;
				gRamAtStopPosition := FALSE;
				gServoRamInterface.Commands.RequestMoveAbs := TRUE;
				ServoRamBusy := TRUE ;
				gRamWaitingOnBox := FALSE;
				state := SERVORAM_TRIGGER_FOLD;
			ELSE
				IF NOT gIO.DIs.SidePickVacuumAchieved THEN
				SideGrabFailAlarm := TRUE;
				state := SERVORAM_ERROR;
			END_IF
		END_IF

		SERVORAM_TRIGGER_FOLD:
			IF gServoRamInterface.Status.ActualPosition > gHMI.Parameters.ServoRamFoldStartPos THEN
				gIO.DOs.FoldingHoldVacuum := TRUE;
				gIO.DOs.LeftSideFoldCylinder := TRUE;
				gIO.DOs.RightSideFoldCylinder := TRUE;
				state := SERVORAM_RELEASE_FOLD;
			END_IF

		SERVORAM_RELEASE_FOLD:
			IF gServoRamInterface.Status.ActualPosition > gHMI.Parameters.ServoRamFoldEndPos THEN
				gIO.DOs.LeftSideFoldCylinder := FALSE;
				gIO.DOs.RightSideFoldCylinder := FALSE;
				state := SERVORAM_MOVE_TO_END;
			END_IF

		SERVORAM_MOVE_TO_END:
			// When the move is complete, check if there is a configured dwell time
			IF gIO.DIs.SidePickVacuumAchieved AND gServoRamInterface.Status.MoveComplete THEN
				gServoRamInterface.Status.MoveComplete := FALSE;
				gRamAtStopPosition := TRUE;
				ServoRamBusy := FALSE;
				gServoRamInterface.Commands.ToMapp.Update := TRUE; //This forces update of the torque limit. This will be cleared automatically
				IF gHMI.Parameters.ServoRamEndDwellTime > 0 THEN
					// If there is a dwell time, execute the dwell
					EndDwellTimer.IN := TRUE;
					state := SERVORAM_DWELL_AT_END;
				ELSE
					// Otherwise, release the vaccuum and move back to the starting position
					gCyclesToFinish := gCyclesToFinish - 1;

					CycleCount := CycleCount + 1;
					LubeCount := LubeCount + 1;
					gIO.DOs.SidePanelVacOn := FALSE;
					gIO.DOs.SidePanelHoldVacuum := FALSE;
					gIO.DOs.FoldingHoldVacuum := FALSE;
					gIO.DOs.LeftSideFoldCylinder := FALSE;
					gIO.DOs.RightSideFoldCylinder := FALSE;
					gServoRamInterface.Parameters.MovementParameters.Position := gHMI.Parameters.ServoRamStartPosition;
					gServoRamInterface.Parameters.MovementParameters.Velocity := gHMI.Parameters.ServoRamNegativeVelocity;
					gServoRamInterface.Commands.RequestMoveAbs := TRUE;
					gRamAtStopPosition := FALSE;
					ServoRamBusy := TRUE;
					gRamWaitingOnBox := TRUE;
					state := SERVORAM_MOVE_TO_START;
				END_IF
				ELSE
					IF NOT gIO.DIs.SidePickVacuumAchieved THEN
					SideGrabFailAlarm := TRUE;
					state := SERVORAM_ERROR;
				END_IF
			END_IF

		SERVORAM_DWELL_AT_END:

			// Wait for the timer to finish
			EndDwellTimer.IN := TRUE;
			IF EndDwellTimer.Q THEN
				gCyclesToFinish := gCyclesToFinish - 1;

				// Release the vacuum and move back to the starting position
				EndDwellTimer.IN := FALSE;
				CycleCount := CycleCount + 1;
				LubeCount := LubeCount + 1;
				gIO.DOs.SidePanelVacOn := FALSE;
				gIO.DOs.SidePanelHoldVacuum := FALSE;
				gIO.DOs.FoldingHoldVacuum := FALSE;
				gIO.DOs.LeftSideFoldCylinder := FALSE;
				gIO.DOs.RightSideFoldCylinder := FALSE;
				gServoRamInterface.Parameters.MovementParameters.Position := gHMI.Parameters.ServoRamStartPosition;
				gServoRamInterface.Parameters.MovementParameters.Velocity := gHMI.Parameters.ServoRamNegativeVelocity;
				gServoRamInterface.Commands.RequestMoveAbs := TRUE;
				gRamAtStopPosition := FALSE;
				ServoRamBusy := TRUE;
				gRamWaitingOnBox := TRUE;
				state := SERVORAM_MOVE_TO_START;
			END_IF

			//these EX states are a copy the states above, but with no actuators being used and no evluation of inputs to know if it is OK to continue
		SERVORAM_MOVE_TO_START_EX:

			IF gServoRamInterface.Status.MoveComplete THEN
				gServoRamInterface.Status.MoveComplete := FALSE;
				ServoRamBusy := FALSE;
				IF NOT ExerciseRam THEN
					state := SERVORAM_IDLE;
				ELSE
					state := SERVORAM_PICK_SIDES_EX;
				END_IF

			END_IF

		SERVORAM_PICK_SIDES_EX:
			SidePickTimer.IN := TRUE;
			// Wait for the side pick timer, then retract the side pick
			IF SidePickTimer.Q THEN
				SidePickRetractTimer.IN := TRUE;
			END_IF
			// When the side pick is retracted, check for side panels
			IF SidePickRetractTimer.Q THEN
				SidePickTimer.IN := FALSE;
				SidePickRetractTimer.IN := FALSE;
				state := SERVORAM_CHECK_FOR_SIDES_EX;
			END_IF

		SERVORAM_CHECK_FOR_SIDES_EX:
			// If the side pick has vacuum, then the sides were picked, move to middle position
			gServoRamInterface.Parameters.MovementParameters.Position := gHMI.Parameters.ServoRamMiddlePosition;
			gServoRamInterface.Parameters.MovementParameters.Velocity := gHMI.Parameters.ServoRamSideFormingVelocity;
			gServoRamInterface.Commands.RequestMoveAbs := TRUE;
			state := SERVORAM_MOVE_TO_MIDDLE_EX;

		SERVORAM_MOVE_TO_MIDDLE_EX:
			// When the ram gets to the middle position, extend the folders
			IF gServoRamInterface.Status.MoveComplete THEN
				gServoRamInterface.Status.MoveComplete := FALSE;
				state := SERVORAM_FOLD_SIDES_EX;
			END_IF

		SERVORAM_FOLD_SIDES_EX:
			SideFoldTimer.IN := TRUE;
			// Wait for the side fold timer, then retract the side folders
			IF SideFoldTimer.Q THEN
				SideFoldRetractTimer.IN := TRUE;
			END_IF
			// When the side fold is retracted, check that the fold was successful
			IF SideFoldRetractTimer.Q THEN
				state := SERVORAM_CHECK_FOR_FOLDS_EX;
			END_IF

		SERVORAM_CHECK_FOR_FOLDS_EX:
			state := SERVORAM_WAITING_ON_BOX_EX;

		SERVORAM_WAITING_ON_BOX_EX:
			RamDelayTimer.IN := TRUE;
			// When the delay finishes, move the ram to the end position
			IF RamDelayTimer.Q THEN
				gServoRamInterface.Parameters.MovementParameters.Position := gHMI.Parameters.ServoRamEndPosition;
				gServoRamInterface.Parameters.MovementParameters.Velocity := gHMI.Parameters.ServoRamBoxFormingVelocity;
				gServoRamInterface.Commands.RequestMoveAbs := TRUE;
				state := SERVORAM_MOVE_TO_END_EX;
			END_IF

		SERVORAM_MOVE_TO_END_EX:
			// When the move is complete, check if there is a configured dwell time
			IF gServoRamInterface.Status.MoveComplete THEN
				gServoRamInterface.Status.MoveComplete := FALSE;
				IF gHMI.Parameters.ServoRamEndDwellTime > 0 THEN
					// If there is a dwell time, execute the dwell
					EndDwellTimer.IN := TRUE;
					state := SERVORAM_DWELL_AT_END_EX;
				ELSE
					// Otherwise, release the vaccuum and move back to the starting position
					CycleCount := CycleCount + 1;
					LubeCount := LubeCount + 1;
					gServoRamInterface.Parameters.MovementParameters.Position := gHMI.Parameters.ServoRamStartPosition;
					gServoRamInterface.Parameters.MovementParameters.Velocity := gHMI.Parameters.ServoRamNegativeVelocity;
					gServoRamInterface.Commands.RequestMoveAbs := TRUE;
					state := SERVORAM_MOVE_TO_START_EX;
				END_IF
			END_IF

		SERVORAM_DWELL_AT_END_EX:

			// Wait for the timer to finish
			EndDwellTimer.IN := TRUE;
			IF EndDwellTimer.Q THEN
				// Release the vacuum and move back to the starting position
				EndDwellTimer.IN := FALSE;
				CycleCount := CycleCount + 1;
				LubeCount := LubeCount + 1;
				gServoRamInterface.Parameters.MovementParameters.Position := gHMI.Parameters.ServoRamStartPosition;
				gServoRamInterface.Parameters.MovementParameters.Velocity := gHMI.Parameters.ServoRamNegativeVelocity;
				gServoRamInterface.Commands.RequestMoveAbs := TRUE;
				state := SERVORAM_MOVE_TO_START_EX;
			END_IF

		SERVORAM_ERROR:

			gCyclesToFinish := 0;

			ServoRamAutoHome := FALSE;
			gServoRamInterface.Status.MoveComplete := FALSE;
			gHMI.Commands.CycleServoRam := FALSE;
			ServoRamBusy := FALSE;
			ServoRamAutoHome := FALSE;
			gIO.DOs.SidePanelHoldVacuum := FALSE;
			gIO.DOs.LeftSideFoldCylinder := FALSE;
			gIO.DOs.RightSideFoldCylinder := FALSE;
			gIO.DOs.SidePickCylinder := FALSE;
			gIO.DOs.SidePanelHoldVacuum := FALSE;
			gIO.DOs.BodyVacuumOn := FALSE;
			gIO.DOs.FoldingHoldVacuum := FALSE;
			gRamWaitingOnBox := FALSE;

			IF (gNumActiveAlarms = 0) THEN
				SideFailureCount := 0;
				FoldFailureCount := 0;
				state := SERVORAM_WAIT_FOR_HOME;
			END_IF

	END_CASE;

	// FUB Calls
	EndDwellTimer.PT := gHMI.Parameters.ServoRamEndDwellTime; //Use existing dwell time from HMI
	EndDwellTimer();
	SidePickTimer.PT := gHMI.Parameters.ServoRamSidePickTime;
	SidePickTimer();
	SidePickRetractTimer.PT := gHMI.Parameters.ServoRamSidePickRetractTime;
	SidePickRetractTimer();
	SideFoldTimer.PT := gHMI.Parameters.ServoRamSideFoldTime;
	SideFoldTimer();
	SideFoldRetractTimer.PT := gHMI.Parameters.ServoRamSideFoldRetractTime;
	SideFoldRetractTimer();
	RamDelayTimer.PT := gHMI.Parameters.RamDelay;
	RamDelayTimer();
	ResetTimeoutTimer.PT := gHMI.Parameters.ServoRamTimeoutTime;
	ResetTimeoutTimer();

END_PROGRAM

PROGRAM _EXIT
				(* Insert code here *)

END_PROGRAM
```
